// TIA Portal V20 export
FUNCTION_BLOCK "CallInterfaceSignals"   // FB38, LAD
TITLE = CallInterfaceSignals
AUTHOR : SICAR
FAMILY : Diag
VERSION : 1.0
// The block serves as a calling interface of the block “InterfaceSignalsBool“. The block is designed as function block in order to implement the block calls as multi-instances.
// stored: IsIECCheckEnabled true, MemoryReserve 100, SetENOAutomatically true
   VAR
      statReadValueHmi : Bool;   // HMI: Read value signal
      statSelectSignalsHmi : USInt := 1;   // HMI: Selected interface signals (1..16)
      statSelectSignalsOld { ExternalAccessible := 'False'; ExternalVisible := 'False'; ExternalWritable := 'False'} : USInt;   // Old value: Selected interface signals
      statRisEdgeReadName { ExternalAccessible := 'False'; ExternalVisible := 'False'; ExternalWritable := 'False'} : Bool;   // Rising edge
      statPosPulseReadName : Bool;   // Positive pulse
      statInterfaceSignalsHmi : Array[0..100] of "typeInterfaceSignalsHmi";   // HMI: Description, value and symbolic name
      instSignals1Left { ExternalAccessible := 'False'; ExternalVisible := 'False'; ExternalWritable := 'False'} : "LAF_InterfaceSignalsBool";   // interface signals screen 1 left
      instSignals1Right { ExternalAccessible := 'False'; ExternalVisible := 'False'; ExternalWritable := 'False'} : "LAF_InterfaceSignalsBool";   // interface signals screen 1 right
      instSignals2Left { ExternalAccessible := 'False'; ExternalVisible := 'False'; ExternalWritable := 'False'} : "LAF_InterfaceSignalsBool";   // interface signals screen 2 left
      instSignals2Right { ExternalAccessible := 'False'; ExternalVisible := 'False'; ExternalWritable := 'False'} : "LAF_InterfaceSignalsBool";   // interface signals screen 2 right
      instSignals3Left { ExternalAccessible := 'False'; ExternalVisible := 'False'; ExternalWritable := 'False'} : "LAF_InterfaceSignalsBool";   // interface signals screen 3 left
      instSignals3Right { ExternalAccessible := 'False'; ExternalVisible := 'False'; ExternalWritable := 'False'} : "LAF_InterfaceSignalsBool";   // interface signals screen 3 right
      instSignals4Left { ExternalAccessible := 'False'; ExternalVisible := 'False'; ExternalWritable := 'False'} : "LAF_InterfaceSignalsBool";   // interface signals screen 4 left
      instSignals4Right { ExternalAccessible := 'False'; ExternalVisible := 'False'; ExternalWritable := 'False'} : "LAF_InterfaceSignalsBool";   // interface signals screen 4 right
      instSignals5Left { ExternalAccessible := 'False'; ExternalVisible := 'False'; ExternalWritable := 'False'} : "LAF_InterfaceSignalsBool";   // interface signals screen 5 left
      instSignals5Right { ExternalAccessible := 'False'; ExternalVisible := 'False'; ExternalWritable := 'False'} : "LAF_InterfaceSignalsBool";   // interface signals screen 5 right
      instSignals6Left { S7_SetPoint := 'True'} : "LAF_InterfaceSignalsBool";   // interface signals screen 6 left
      instSignals6Right { S7_SetPoint := 'True'} : "LAF_InterfaceSignalsBool";   // interface signals screen 6 right
      instSignals7Left { S7_SetPoint := 'True'} : "LAF_InterfaceSignalsBool";   // interface signals screen 7 left
      instSignals7Right { S7_SetPoint := 'True'} : "LAF_InterfaceSignalsBool";   // interface signals screen 7 right
      instSignals8Left { S7_SetPoint := 'True'} : "LAF_InterfaceSignalsBool";   // interface signals screen 8 left
      instSignals8Right { S7_SetPoint := 'True'} : "LAF_InterfaceSignalsBool";   // interface signals screen 8 right
      instSignals9Left { S7_SetPoint := 'True'} : "LAF_InterfaceSignalsBool";   // interface signals screen 9 left
      instSignals9Right { S7_SetPoint := 'True'} : "LAF_InterfaceSignalsBool";   // interface signals screen 9 right
      instSignals10Left_ { S7_SetPoint := 'True'} : "LAF_InterfaceSignalsBool";   // interface signals screen 10 left
      instSignals10Right { S7_SetPoint := 'True'} : "LAF_InterfaceSignalsBool";   // interface signals screen 10 right
      instSignals11Left { S7_SetPoint := 'True'} : "LAF_InterfaceSignalsBool";   // interface signals screen 11 left
      instSignals11Right { S7_SetPoint := 'True'} : "LAF_InterfaceSignalsBool";   // interface signals screen 11 right
      instSignals12Left { S7_SetPoint := 'True'} : "LAF_InterfaceSignalsBool";   // interface signals screen 12 left
      instSignals12Right { S7_SetPoint := 'True'} : "LAF_InterfaceSignalsBool";   // interface signals screen 12 right
      instSignals13Left { S7_SetPoint := 'True'} : "LAF_InterfaceSignalsBool";   // interface signals screen 13 left
      instSignals13Right { S7_SetPoint := 'True'} : "LAF_InterfaceSignalsBool";   // interface signals screen 13 right
      instSignals14Left { S7_SetPoint := 'True'} : "LAF_InterfaceSignalsBool";   // interface signals screen 14 left
      instSignals14Right { S7_SetPoint := 'True'} : "LAF_InterfaceSignalsBool";   // interface signals screen 14 right
      instSignals15Left { S7_SetPoint := 'True'} : "LAF_InterfaceSignalsBool";   // interface signals screen 15 left
      instSignals15Right { S7_SetPoint := 'True'} : "LAF_InterfaceSignalsBool";   // interface signals screen 15 right
      instSignals16Left { S7_SetPoint := 'True'} : "LAF_InterfaceSignalsBool";   // interface signals screen 16 left
      instSignals16Right { S7_SetPoint := 'True'} : "LAF_InterfaceSignalsBool";   // interface signals screen 16 right
      instSignals17Left { S7_SetPoint := 'True'} : "LAF_InterfaceSignalsBool";   // interface signals screen 17 left
      instSignals17Right { S7_SetPoint := 'True'} : "LAF_InterfaceSignalsBool";   // interface signals screen 17 right
      instSignals18Left { S7_SetPoint := 'True'} : "LAF_InterfaceSignalsBool";   // interface signals screen 18 left
      instSignals18Right { S7_SetPoint := 'True'} : "LAF_InterfaceSignalsBool";   // interface signals screen 18 right
      instSignals19Left { S7_SetPoint := 'True'} : "LAF_InterfaceSignalsBool";   // interface signals screen 19 left
      instSignals19Right { S7_SetPoint := 'True'} : "LAF_InterfaceSignalsBool";   // interface signals screen 19 right
      instSignals20Left { S7_SetPoint := 'True'} : "LAF_InterfaceSignalsBool";   // interface signals screen 20 left
      instSignals20Right { S7_SetPoint := 'True'} : "LAF_InterfaceSignalsBool";   // interface signals screen 20 right
      instSignals21Left { S7_SetPoint := 'True'} : "LAF_InterfaceSignalsBool";   // interface signals screen 21 left
      instSignals21Right { S7_SetPoint := 'True'} : "LAF_InterfaceSignalsBool";   // interface signals screen 21 right
      instSignals22Left { S7_SetPoint := 'True'} : "LAF_InterfaceSignalsBool";   // interface signals screen 22 left
      instSignals22Right { S7_SetPoint := 'True'} : "LAF_InterfaceSignalsBool";   // interface signals screen 22 right
      instSignals23Left { S7_SetPoint := 'True'} : "LAF_InterfaceSignalsBool";   // interface signals screen 23 left
      instSignals23Right { S7_SetPoint := 'True'} : "LAF_InterfaceSignalsBool";   // interface signals screen 23 right
      instSignals24Left { S7_SetPoint := 'True'} : "LAF_InterfaceSignalsBool";   // interface signals screen 24 left
      instSignals24Right { S7_SetPoint := 'True'} : "LAF_InterfaceSignalsBool";   // interface signals screen 24 right
      instSignals25Left { S7_SetPoint := 'True'} : "LAF_InterfaceSignalsBool";   // interface signals screen 25 left
      instSignals25Right { S7_SetPoint := 'True'} : "LAF_InterfaceSignalsBool";   // interface signals screen 25 right
      instSignals26Left { S7_SetPoint := 'True'} : "LAF_InterfaceSignalsBool";   // interface signals screen 26 left
      instSignals26Right { S7_SetPoint := 'True'} : "LAF_InterfaceSignalsBool";   // interface signals screen 26 right
      instSignals27Left { S7_SetPoint := 'True'} : "LAF_InterfaceSignalsBool";   // interface signals screen 27 left
      instSignals27Right { S7_SetPoint := 'True'} : "LAF_InterfaceSignalsBool";   // interface signals screen 27 right
      instSignals28Left { S7_SetPoint := 'True'} : "LAF_InterfaceSignalsBool";   // interface signals screen 28 left
      instSignals28Right { S7_SetPoint := 'True'} : "LAF_InterfaceSignalsBool";   // interface signals screen 28 right
      instSignals29Left { S7_SetPoint := 'True'} : "LAF_InterfaceSignalsBool";   // interface signals screen 29 left
      instSignals29Right { S7_SetPoint := 'True'} : "LAF_InterfaceSignalsBool";   // interface signals screen 29 right
      instSignals30Left { S7_SetPoint := 'True'} : "LAF_InterfaceSignalsBool";   // interface signals screen 30 left
      instSignals30Right { S7_SetPoint := 'True'} : "LAF_InterfaceSignalsBool";   // interface signals screen 30 right
      instSignals31Left { S7_SetPoint := 'True'} : "LAF_InterfaceSignalsBool";   // interface signals screen 31 left
      instSignals31Right { S7_SetPoint := 'True'} : "LAF_InterfaceSignalsBool";   // interface signals screen 31 right
      instSignals32Left { S7_SetPoint := 'True'} : "LAF_InterfaceSignalsBool";   // interface signals screen 32 left
      instSignals32Right { S7_SetPoint := 'True'} : "LAF_InterfaceSignalsBool";   // interface signals screen 32 right
      instSignals33Left { S7_SetPoint := 'True'} : "LAF_InterfaceSignalsBool";   // interface signals screen 33 left
      instSignals33Right { S7_SetPoint := 'True'} : "LAF_InterfaceSignalsBool";   // interface signals screen 33 right
      instSignals34Left { S7_SetPoint := 'True'} : "LAF_InterfaceSignalsBool";   // interface signals screen 34 left
      instSignals34Right { S7_SetPoint := 'True'} : "LAF_InterfaceSignalsBool";   // interface signals screen 34 right
      instSignals35Left { S7_SetPoint := 'True'} : "LAF_InterfaceSignalsBool";   // interface signals screen 35 left
      instSignals35Right { S7_SetPoint := 'True'} : "LAF_InterfaceSignalsBool";   // interface signals screen 35 right
      instSignals36Left { S7_SetPoint := 'True'} : "LAF_InterfaceSignalsBool";   // interface signals screen 36 left
      instSignals36Right { S7_SetPoint := 'True'} : "LAF_InterfaceSignalsBool";   // interface signals screen 36 right
      instSignals37Left { S7_SetPoint := 'True'} : "LAF_InterfaceSignalsBool";   // interface signals screen 37 left
      instSignals37Right { S7_SetPoint := 'True'} : "LAF_InterfaceSignalsBool";   // interface signals screen 37 right
      instSignals38Left { S7_SetPoint := 'True'} : "LAF_InterfaceSignalsBool";   // interface signals screen 38 left
      instSignals38Right { S7_SetPoint := 'True'} : "LAF_InterfaceSignalsBool";   // interface signals screen 38 right
      instSignals39Left { S7_SetPoint := 'True'} : "LAF_InterfaceSignalsBool";   // interface signals screen 39 left
      instSignals39Right { S7_SetPoint := 'True'} : "LAF_InterfaceSignalsBool";   // interface signals screen 39 right
      instSignals40Left { S7_SetPoint := 'True'} : "LAF_InterfaceSignalsBool";   // interface signals screen 40 left
      instSignals40Right { S7_SetPoint := 'True'} : "LAF_InterfaceSignalsBool";   // interface signals screen 40 right
      instSignals41Left { S7_SetPoint := 'True'} : "LAF_InterfaceSignalsBool";   // interface signals screen 41 left
      instSignals41Right { S7_SetPoint := 'True'} : "LAF_InterfaceSignalsBool";   // interface signals screen 41 right
      instSignals42Left { S7_SetPoint := 'True'} : "LAF_InterfaceSignalsBool";   // interface signals screen 42 left
      instSignals42Right { S7_SetPoint := 'True'} : "LAF_InterfaceSignalsBool";   // interface signals screen 42 right
      instSignals43Left { S7_SetPoint := 'True'} : "LAF_InterfaceSignalsBool";   // interface signals screen 43 left
      instSignals43Right { S7_SetPoint := 'True'} : "LAF_InterfaceSignalsBool";   // interface signals screen 43 right
      instSignals44Left { S7_SetPoint := 'True'} : "LAF_InterfaceSignalsBool";   // interface signals screen 44 left
      instSignals44Right { S7_SetPoint := 'True'} : "LAF_InterfaceSignalsBool";   // interface signals screen 44 right
      instSignals45Left { S7_SetPoint := 'True'} : "LAF_InterfaceSignalsBool";   // interface signals screen 45 left
      instSignals45Right { S7_SetPoint := 'True'} : "LAF_InterfaceSignalsBool";   // interface signals screen 45 right
      instSignals46Left { S7_SetPoint := 'True'} : "LAF_InterfaceSignalsBool";   // interface signals screen 46 left
      instSignals46Right { S7_SetPoint := 'True'} : "LAF_InterfaceSignalsBool";   // interface signals screen 46 right
      instSignals47Left { S7_SetPoint := 'True'} : "LAF_InterfaceSignalsBool";   // interface signals screen 47 left
      instSignals47Right { S7_SetPoint := 'True'} : "LAF_InterfaceSignalsBool";   // interface signals screen 47 right
      instSignals48Left { S7_SetPoint := 'True'} : "LAF_InterfaceSignalsBool";   // interface signals screen 48 left
      instSignals48Right { S7_SetPoint := 'True'} : "LAF_InterfaceSignalsBool";   // interface signals screen 48 right
      instSignals49Left { S7_SetPoint := 'True'} : "LAF_InterfaceSignalsBool";   // interface signals screen 49 left
      instSignals49Right { S7_SetPoint := 'True'} : "LAF_InterfaceSignalsBool";   // interface signals screen 49 right
      instSignals50Left { S7_SetPoint := 'True'} : "LAF_InterfaceSignalsBool";   // interface signals screen 50 left
      instSignals50Right { S7_SetPoint := 'True'} : "LAF_InterfaceSignalsBool";   // interface signals screen 50 right
      instSignals51Left { S7_SetPoint := 'True'} : "LAF_InterfaceSignalsBool";   // interface signals screen 51 left
      instSignals51Right { S7_SetPoint := 'True'} : "LAF_InterfaceSignalsBool";   // interface signals screen 51 right
      instSignals52Left { S7_SetPoint := 'True'} : "LAF_InterfaceSignalsBool";   // interface signals screen 52 left
      instSignals52Right { S7_SetPoint := 'True'} : "LAF_InterfaceSignalsBool";   // interface signals screen 52 right
      instSignals53Left { S7_SetPoint := 'True'} : "LAF_InterfaceSignalsBool";   // interface signals screen 53 left
      instSignals53Right { S7_SetPoint := 'True'} : "LAF_InterfaceSignalsBool";   // interface signals screen 53 right
      instSignals54Left { S7_SetPoint := 'True'} : "LAF_InterfaceSignalsBool";   // interface signals screen 54 left
      instSignals54Right { S7_SetPoint := 'True'} : "LAF_InterfaceSignalsBool";   // interface signals screen 54 right
      instSignals55Left { S7_SetPoint := 'True'} : "LAF_InterfaceSignalsBool";   // interface signals screen 55 left
      instSignals55Right { S7_SetPoint := 'True'} : "LAF_InterfaceSignalsBool";   // interface signals screen 55 right
      instSignals56Left { S7_SetPoint := 'True'} : "LAF_InterfaceSignalsBool";   // interface signals screen 56 left
      instSignals56Right { S7_SetPoint := 'True'} : "LAF_InterfaceSignalsBool";   // interface signals screen 56 right
      instSignals57Left { S7_SetPoint := 'True'} : "LAF_InterfaceSignalsBool";   // interface signals screen 57 left
      instSignals57Right { S7_SetPoint := 'True'} : "LAF_InterfaceSignalsBool";   // interface signals screen 57 right
      instSignals58Left { S7_SetPoint := 'True'} : "LAF_InterfaceSignalsBool";   // interface signals screen 58 left
      instSignals58Right { S7_SetPoint := 'True'} : "LAF_InterfaceSignalsBool";   // interface signals screen 58 right
      instSignals59Left { S7_SetPoint := 'True'} : "LAF_InterfaceSignalsBool";   // interface signals screen 59 left
      instSignals59Right { S7_SetPoint := 'True'} : "LAF_InterfaceSignalsBool";   // interface signals screen 59 right
      instSignals60Left { S7_SetPoint := 'True'} : "LAF_InterfaceSignalsBool";   // interface signals screen 60 left
      instSignals60Right { S7_SetPoint := 'True'} : "LAF_InterfaceSignalsBool";   // interface signals screen 60 right
      instSignals61Left { S7_SetPoint := 'True'} : "LAF_InterfaceSignalsBool";   // interface signals screen 61 left
      instSignals61Right { S7_SetPoint := 'True'} : "LAF_InterfaceSignalsBool";   // interface signals screen 61 right
      instSignals62Left { S7_SetPoint := 'True'} : "LAF_InterfaceSignalsBool";   // interface signals screen 62 left
      instSignals62Right { S7_SetPoint := 'True'} : "LAF_InterfaceSignalsBool";   // interface signals screen 62 right
      instSignals63Left { S7_SetPoint := 'True'} : "LAF_InterfaceSignalsBool";   // interface signals screen 63 left
      instSignals63Right { S7_SetPoint := 'True'} : "LAF_InterfaceSignalsBool";   // interface signals screen 63 right
      instSignals64Left { S7_SetPoint := 'True'} : "LAF_InterfaceSignalsBool";   // interface signals screen 64 left
      instSignals64Right { S7_SetPoint := 'True'} : "LAF_InterfaceSignalsBool";   // interface signals screen 64 right
      instSignals65Left { S7_SetPoint := 'True'} : "LAF_InterfaceSignalsBool";   // interface signals screen 65 left
      instSignals65Right { S7_SetPoint := 'True'} : "LAF_InterfaceSignalsBool";   // interface signals screen 65 right
      instSignals66Left { S7_SetPoint := 'True'} : "LAF_InterfaceSignalsBool";   // interface signals screen 66 left
      instSignals66Right { S7_SetPoint := 'True'} : "LAF_InterfaceSignalsBool";   // interface signals screen 66 right
      instSignals67Left { S7_SetPoint := 'True'} : "LAF_InterfaceSignalsBool";   // interface signals screen 67 left
      instSignals67Right { S7_SetPoint := 'True'} : "LAF_InterfaceSignalsBool";   // interface signals screen 67 right
      instSignals68Left { S7_SetPoint := 'True'} : "LAF_InterfaceSignalsBool";   // interface signals screen 68 left
      instSignals68Right { S7_SetPoint := 'True'} : "LAF_InterfaceSignalsBool";   // interface signals screen 68 right
      instSignals69Left { S7_SetPoint := 'True'} : "LAF_InterfaceSignalsBool";   // interface signals screen 69 left
      instSignals69Right { S7_SetPoint := 'True'} : "LAF_InterfaceSignalsBool";   // interface signals screen 69 right
      instSignals70Left { S7_SetPoint := 'True'} : "LAF_InterfaceSignalsBool";   // interface signals screen 70 left
      instSignals70Right { S7_SetPoint := 'True'} : "LAF_InterfaceSignalsBool";   // interface signals screen 70 right
      instSignals71Left { S7_SetPoint := 'True'} : "LAF_InterfaceSignalsBool";   // interface signals screen 71 left
      instSignals71Right { S7_SetPoint := 'True'} : "LAF_InterfaceSignalsBool";   // interface signals screen 71 right
      instSignals72Left { S7_SetPoint := 'True'} : "LAF_InterfaceSignalsBool";   // interface signals screen 72 left
      instSignals72Right { S7_SetPoint := 'True'} : "LAF_InterfaceSignalsBool";   // interface signals screen 72 right
      instSignals73Left { S7_SetPoint := 'True'} : "LAF_InterfaceSignalsBool";   // interface signals screen 73 left
      instSignals73Right { S7_SetPoint := 'True'} : "LAF_InterfaceSignalsBool";   // interface signals screen 73 right
      instSignals74Left { S7_SetPoint := 'True'} : "LAF_InterfaceSignalsBool";   // interface signals screen 74 left
      instSignals74Right { S7_SetPoint := 'True'} : "LAF_InterfaceSignalsBool";   // interface signals screen 74 right
      instSignals75Left { S7_SetPoint := 'True'} : "LAF_InterfaceSignalsBool";   // interface signals screen 75 left
      instSignals75Right { S7_SetPoint := 'True'} : "LAF_InterfaceSignalsBool";   // interface signals screen 75 right
      instSignals76Left { S7_SetPoint := 'True'} : "LAF_InterfaceSignalsBool";   // interface signals screen 76 left
      instSignals76Right { S7_SetPoint := 'True'} : "LAF_InterfaceSignalsBool";   // interface signals screen 76 right
   END_VAR
   VAR_TEMP
      tempLoopCounter : DInt;   // temp. Loop Counter
   END_VAR
   VAR_TEMP   // added for the SCL form of the ladder/FBD networks
      _w1 : Bool;
   END_VAR
BEGIN

REGION Network 1: BLOCK INFO HEADER
   // SIEMENS AG / (c)Copyright 2023
   // ------------------------------------------------------------------------------
   // Title:            CallInterfaceSignals (FB38)
   // Comment/Function: The block serves as a calling interface of the block “InterfaceSignalsBool“. The block is designed as function block in order to implement the block calls as multi-instances. 
   // Library/Family:   Diag
   // Author:           SICAR
   // Tested with:      ---
   // Engineering:      TIA Portal V19
   // Restrictions:     -
   // Requirements:     ---
   // ------------------------------------------------------------------------------
   // Change log table:
   // Version  | Date       | Expert in charge       | Changes applied
   // ---------|------------|------------------------|------------------------------
   // 01.00.00 | 11.12.2023 | SICAR
   //                         First released version
END_REGION

REGION Network 2: DESCRIPTION
   // Function block and corresponding WinCC screen are prepared for 16 data sets (“InterfaceSignals01“ through .”InterfaceSignals16“) with 32 Boolean signals each.  
   // 
   // **PLC-Data types**   
   // 
   // * LSicar_typeInterfaceSignalsBool 
   // * LSicar _typeInterfaceSignals 
   // * typeInterfaceSignalsHmi 
   // 
   // **WinCC-Faceplate**  
   // 
   // <None> 
   // 
   // **WinCC Diagnostic screen**   
   // 
   // See: ..\Library Types\LSicar_InterfaceSignalsBool.pdf  
   // 
   // **Block call example** 
   // 
   // View in ladder-logic (LAD), without parameter settings.  
   // An executable program call is available in the “SICAR-Startup” project.  
   // 
   // **Calling interface**  
   // 
   // The block is be called once in the cyclic program.  
   // 
   // **Internally used „Extended instructions / blocks“**  
   // 
   // See: ..\Library Types\LSicar_InterfaceSignalsBool.pdf
END_REGION

REGION Network 3: Initialization Loop_1
   // Preset the loop index
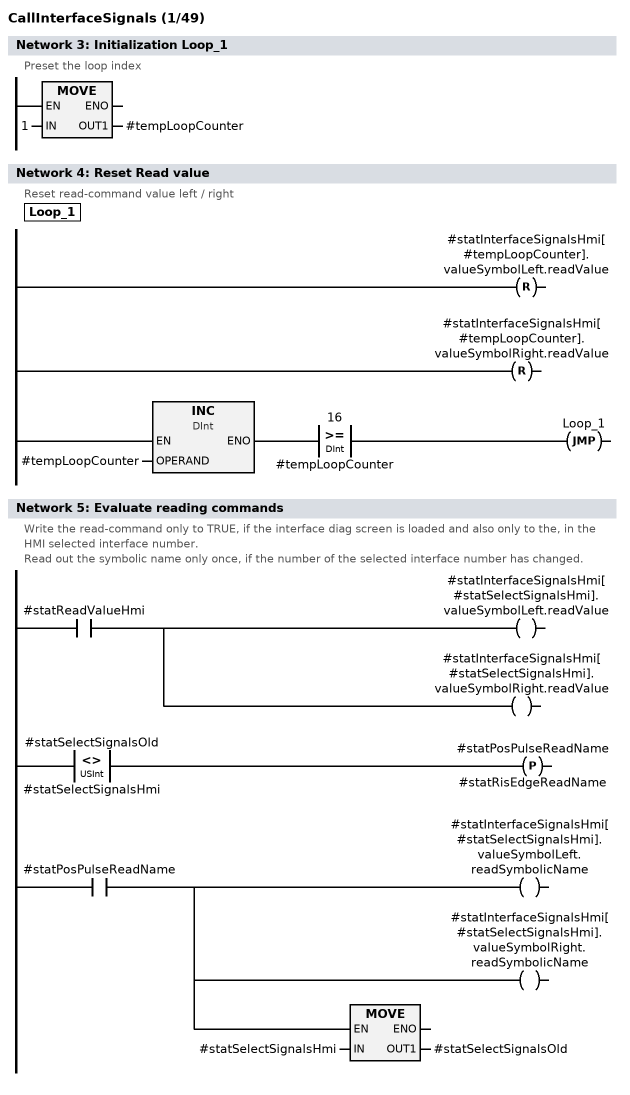
   RUNG wire#powerrail
      Move(in := 1, out1 => #tempLoopCounter)
   END_RUNG
   // the same network as SCL:
   #tempLoopCounter := 1;
END_REGION

REGION Network 4: Reset Read value
   // Reset read-command value left / right
   Label( Loop_1 )
   RUNG wire#powerrail
      R_Coil( #statInterfaceSignalsHmi[#tempLoopCounter].valueSymbolLeft.readValue )
   END_RUNG
   RUNG wire#powerrail
      R_Coil( #statInterfaceSignalsHmi[#tempLoopCounter].valueSymbolRight.readValue )
   END_RUNG
   RUNG wire#powerrail
      { S7_Templates := "DestType := DInt" } Inc( #tempLoopCounter )
      { S7_Templates := "SrcType := DInt" } GE_Contact(in1 := 16, in2 := #tempLoopCounter)
      JumpCoil( Loop_1 )
   END_RUNG
   // the same network as SCL:
   Loop_1:
   #statInterfaceSignalsHmi[#tempLoopCounter].valueSymbolLeft.readValue := FALSE;
   #statInterfaceSignalsHmi[#tempLoopCounter].valueSymbolRight.readValue := FALSE;
   #tempLoopCounter := #tempLoopCounter + 1;
   IF 16 >= #tempLoopCounter THEN GOTO Loop_1; END_IF;
END_REGION

REGION Network 5: Evaluate reading commands
   // Write the read-command only to TRUE, if the interface diag screen is loaded and also only to the, in the HMI selected interface number.
   // Read out the symbolic name only once, if the number of the selected interface number has changed.
   #statInterfaceSignalsHmi[#statSelectSignalsHmi].valueSymbolLeft.readValue := #statReadValueHmi;
   #statInterfaceSignalsHmi[#statSelectSignalsHmi].valueSymbolRight.readValue := #statReadValueHmi;
   #_w1 := #statSelectSignalsOld <> #statSelectSignalsHmi;
   #statPosPulseReadName := #_w1 AND NOT #statRisEdgeReadName;   // rising edge
   #statRisEdgeReadName := #_w1;
   #statInterfaceSignalsHmi[#statSelectSignalsHmi].valueSymbolLeft.readSymbolicName := #statPosPulseReadName;
   #statInterfaceSignalsHmi[#statSelectSignalsHmi].valueSymbolRight.readSymbolicName := #statPosPulseReadName;
   IF #statPosPulseReadName THEN #statSelectSignalsOld := #statSelectSignalsHmi; END_IF;
END_REGION

REGION Network 6: Interface Signals 01 BA030
   // Call the interface signals bool blocks of system tags
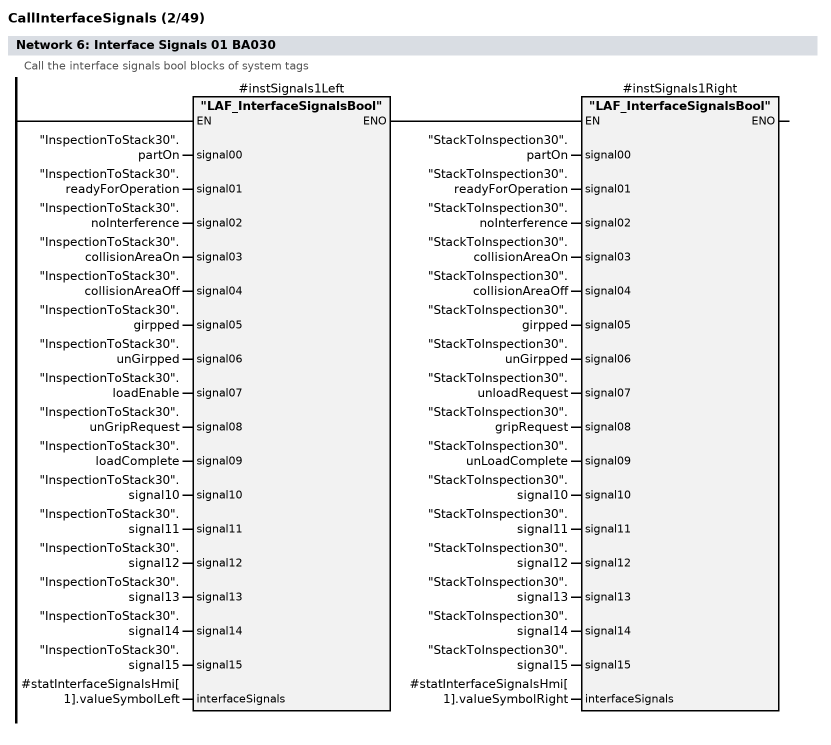
   RUNG wire#powerrail
      #instSignals1Left(signal00 := "InspectionToStack30".partOn, signal01 := "InspectionToStack30".readyForOperation, signal02 := "InspectionToStack30".noInterference, signal03 := "InspectionToStack30".collisionAreaOn, signal04 := "InspectionToStack30".collisionAreaOff, signal05 := "InspectionToStack30".girpped, signal06 := "InspectionToStack30".unGirpped, signal07 := "InspectionToStack30".loadEnable, signal08 := "InspectionToStack30".unGripRequest, signal09 := "InspectionToStack30".loadComplete, signal10 := "InspectionToStack30".signal10, signal11 := "InspectionToStack30".signal11, signal12 := "InspectionToStack30".signal12, signal13 := "InspectionToStack30".signal13, signal14 := "InspectionToStack30".signal14, signal15 := "InspectionToStack30".signal15, interfaceSignals := #statInterfaceSignalsHmi[1].valueSymbolLeft)
      #instSignals1Right(signal00 := "StackToInspection30".partOn, signal01 := "StackToInspection30".readyForOperation, signal02 := "StackToInspection30".noInterference, signal03 := "StackToInspection30".collisionAreaOn, signal04 := "StackToInspection30".collisionAreaOff, signal05 := "StackToInspection30".girpped, signal06 := "StackToInspection30".unGirpped, signal07 := "StackToInspection30".unloadRequest, signal08 := "StackToInspection30".gripRequest, signal09 := "StackToInspection30".unLoadComplete, signal10 := "StackToInspection30".signal10, signal11 := "StackToInspection30".signal11, signal12 := "StackToInspection30".signal12, signal13 := "StackToInspection30".signal13, signal14 := "StackToInspection30".signal14, signal15 := "StackToInspection30".signal15, interfaceSignals := #statInterfaceSignalsHmi[1].valueSymbolRight)
   END_RUNG
   // the same network as SCL:
   #instSignals1Left(signal00 := "InspectionToStack30".partOn,   // "LAF_InterfaceSignalsBool"
                     signal01 := "InspectionToStack30".readyForOperation,
                     signal02 := "InspectionToStack30".noInterference,
                     signal03 := "InspectionToStack30".collisionAreaOn,
                     signal04 := "InspectionToStack30".collisionAreaOff,
                     signal05 := "InspectionToStack30".girpped,
                     signal06 := "InspectionToStack30".unGirpped,
                     signal07 := "InspectionToStack30".loadEnable,
                     signal08 := "InspectionToStack30".unGripRequest,
                     signal09 := "InspectionToStack30".loadComplete,
                     signal10 := "InspectionToStack30".signal10,
                     signal11 := "InspectionToStack30".signal11,
                     signal12 := "InspectionToStack30".signal12,
                     signal13 := "InspectionToStack30".signal13,
                     signal14 := "InspectionToStack30".signal14,
                     signal15 := "InspectionToStack30".signal15,
                     interfaceSignals := #statInterfaceSignalsHmi[1].valueSymbolLeft,
                     ENO => #_w1);
   IF #_w1 THEN
       #instSignals1Right(signal00 := "StackToInspection30".partOn,   // "LAF_InterfaceSignalsBool"
                          signal01 := "StackToInspection30".readyForOperation,
                          signal02 := "StackToInspection30".noInterference,
                          signal03 := "StackToInspection30".collisionAreaOn,
                          signal04 := "StackToInspection30".collisionAreaOff,
                          signal05 := "StackToInspection30".girpped,
                          signal06 := "StackToInspection30".unGirpped,
                          signal07 := "StackToInspection30".unloadRequest,
                          signal08 := "StackToInspection30".gripRequest,
                          signal09 := "StackToInspection30".unLoadComplete,
                          signal10 := "StackToInspection30".signal10,
                          signal11 := "StackToInspection30".signal11,
                          signal12 := "StackToInspection30".signal12,
                          signal13 := "StackToInspection30".signal13,
                          signal14 := "StackToInspection30".signal14,
                          signal15 := "StackToInspection30".signal15,
                          interfaceSignals := #statInterfaceSignalsHmi[1].valueSymbolRight);
   END_IF;
END_REGION

REGION Network 7: Interface Signals 02 BA040
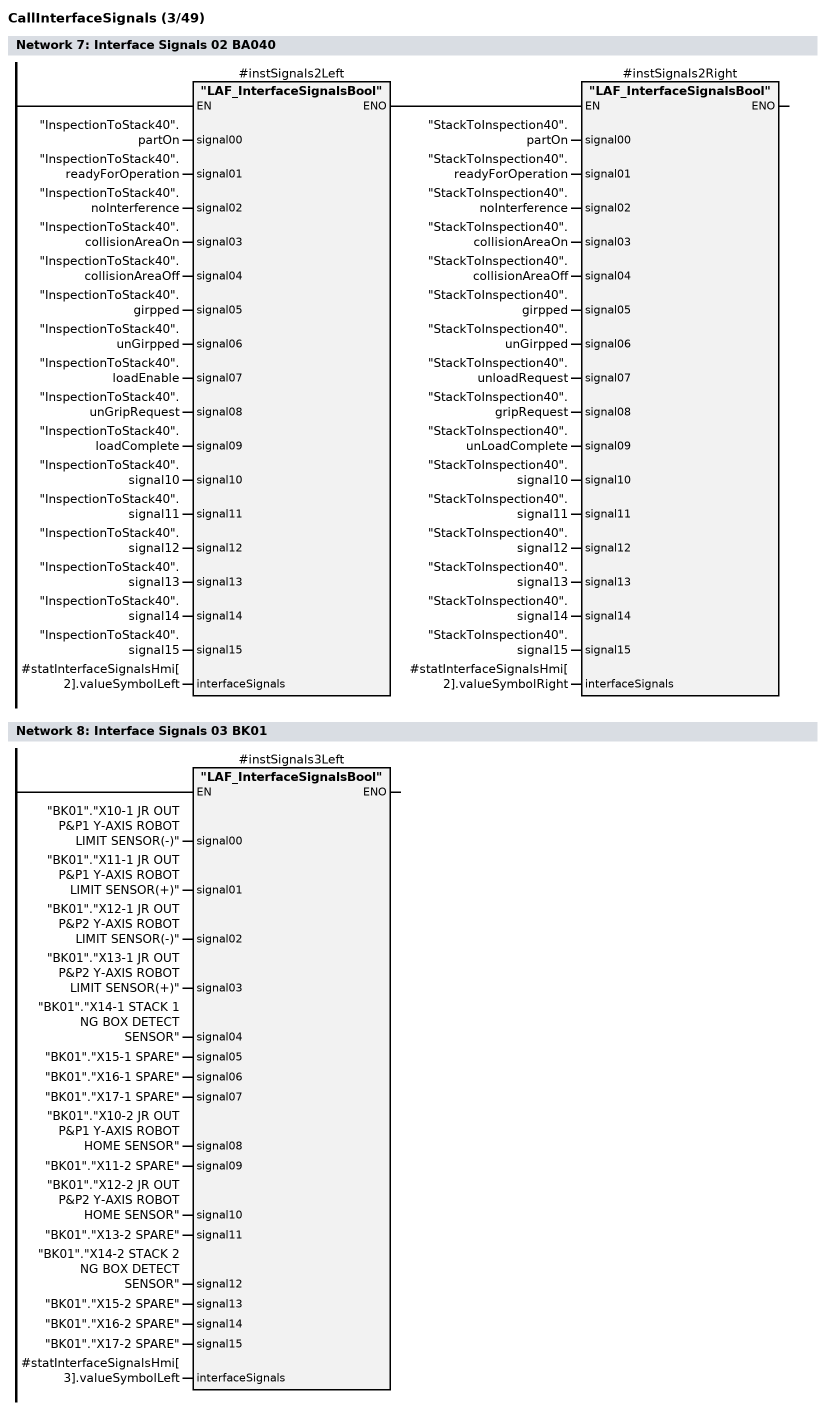
   RUNG wire#powerrail
      #instSignals2Left(signal00 := "InspectionToStack40".partOn, signal01 := "InspectionToStack40".readyForOperation, signal02 := "InspectionToStack40".noInterference, signal03 := "InspectionToStack40".collisionAreaOn, signal04 := "InspectionToStack40".collisionAreaOff, signal05 := "InspectionToStack40".girpped, signal06 := "InspectionToStack40".unGirpped, signal07 := "InspectionToStack40".loadEnable, signal08 := "InspectionToStack40".unGripRequest, signal09 := "InspectionToStack40".loadComplete, signal10 := "InspectionToStack40".signal10, signal11 := "InspectionToStack40".signal11, signal12 := "InspectionToStack40".signal12, signal13 := "InspectionToStack40".signal13, signal14 := "InspectionToStack40".signal14, signal15 := "InspectionToStack40".signal15, interfaceSignals := #statInterfaceSignalsHmi[2].valueSymbolLeft)
      #instSignals2Right(signal00 := "StackToInspection40".partOn, signal01 := "StackToInspection40".readyForOperation, signal02 := "StackToInspection40".noInterference, signal03 := "StackToInspection40".collisionAreaOn, signal04 := "StackToInspection40".collisionAreaOff, signal05 := "StackToInspection40".girpped, signal06 := "StackToInspection40".unGirpped, signal07 := "StackToInspection40".unloadRequest, signal08 := "StackToInspection40".gripRequest, signal09 := "StackToInspection40".unLoadComplete, signal10 := "StackToInspection40".signal10, signal11 := "StackToInspection40".signal11, signal12 := "StackToInspection40".signal12, signal13 := "StackToInspection40".signal13, signal14 := "StackToInspection40".signal14, signal15 := "StackToInspection40".signal15, interfaceSignals := #statInterfaceSignalsHmi[2].valueSymbolRight)
   END_RUNG
   // the same network as SCL:
   #instSignals2Left(signal00 := "InspectionToStack40".partOn,   // "LAF_InterfaceSignalsBool"
                     signal01 := "InspectionToStack40".readyForOperation,
                     signal02 := "InspectionToStack40".noInterference,
                     signal03 := "InspectionToStack40".collisionAreaOn,
                     signal04 := "InspectionToStack40".collisionAreaOff,
                     signal05 := "InspectionToStack40".girpped,
                     signal06 := "InspectionToStack40".unGirpped,
                     signal07 := "InspectionToStack40".loadEnable,
                     signal08 := "InspectionToStack40".unGripRequest,
                     signal09 := "InspectionToStack40".loadComplete,
                     signal10 := "InspectionToStack40".signal10,
                     signal11 := "InspectionToStack40".signal11,
                     signal12 := "InspectionToStack40".signal12,
                     signal13 := "InspectionToStack40".signal13,
                     signal14 := "InspectionToStack40".signal14,
                     signal15 := "InspectionToStack40".signal15,
                     interfaceSignals := #statInterfaceSignalsHmi[2].valueSymbolLeft,
                     ENO => #_w1);
   IF #_w1 THEN
       #instSignals2Right(signal00 := "StackToInspection40".partOn,   // "LAF_InterfaceSignalsBool"
                          signal01 := "StackToInspection40".readyForOperation,
                          signal02 := "StackToInspection40".noInterference,
                          signal03 := "StackToInspection40".collisionAreaOn,
                          signal04 := "StackToInspection40".collisionAreaOff,
                          signal05 := "StackToInspection40".girpped,
                          signal06 := "StackToInspection40".unGirpped,
                          signal07 := "StackToInspection40".unloadRequest,
                          signal08 := "StackToInspection40".gripRequest,
                          signal09 := "StackToInspection40".unLoadComplete,
                          signal10 := "StackToInspection40".signal10,
                          signal11 := "StackToInspection40".signal11,
                          signal12 := "StackToInspection40".signal12,
                          signal13 := "StackToInspection40".signal13,
                          signal14 := "StackToInspection40".signal14,
                          signal15 := "StackToInspection40".signal15,
                          interfaceSignals := #statInterfaceSignalsHmi[2].valueSymbolRight);
   END_IF;
END_REGION

REGION Network 8: Interface Signals 03 BK01
   RUNG wire#powerrail
      #instSignals3Left(signal00 := "BK01"."X10-1 JR OUT P&P1 Y-AXIS ROBOT LIMIT SENSOR(-)", signal01 := "BK01"."X11-1 JR OUT P&P1 Y-AXIS ROBOT LIMIT SENSOR(+)", signal02 := "BK01"."X12-1 JR OUT P&P2 Y-AXIS ROBOT LIMIT SENSOR(-)", signal03 := "BK01"."X13-1 JR OUT P&P2 Y-AXIS ROBOT LIMIT SENSOR(+)", signal04 := "BK01"."X14-1 STACK 1 NG BOX DETECT SENSOR", signal05 := "BK01"."X15-1 SPARE", signal06 := "BK01"."X16-1 SPARE", signal07 := "BK01"."X17-1 SPARE", signal08 := "BK01"."X10-2 JR OUT P&P1 Y-AXIS ROBOT HOME SENSOR", signal09 := "BK01"."X11-2 SPARE", signal10 := "BK01"."X12-2 JR OUT P&P2 Y-AXIS ROBOT HOME SENSOR", signal11 := "BK01"."X13-2 SPARE", signal12 := "BK01"."X14-2 STACK 2 NG BOX DETECT SENSOR", signal13 := "BK01"."X15-2 SPARE", signal14 := "BK01"."X16-2 SPARE", signal15 := "BK01"."X17-2 SPARE", interfaceSignals := #statInterfaceSignalsHmi[3].valueSymbolLeft)
   END_RUNG
   // the same network as SCL:
   #instSignals3Left(signal00 := "BK01"."X10-1 JR OUT P&P1 Y-AXIS ROBOT LIMIT SENSOR(-)",   // "LAF_InterfaceSignalsBool"
                     signal01 := "BK01"."X11-1 JR OUT P&P1 Y-AXIS ROBOT LIMIT SENSOR(+)",
                     signal02 := "BK01"."X12-1 JR OUT P&P2 Y-AXIS ROBOT LIMIT SENSOR(-)",
                     signal03 := "BK01"."X13-1 JR OUT P&P2 Y-AXIS ROBOT LIMIT SENSOR(+)",
                     signal04 := "BK01"."X14-1 STACK 1 NG BOX DETECT SENSOR",
                     signal05 := "BK01"."X15-1 SPARE",
                     signal06 := "BK01"."X16-1 SPARE",
                     signal07 := "BK01"."X17-1 SPARE",
                     signal08 := "BK01"."X10-2 JR OUT P&P1 Y-AXIS ROBOT HOME SENSOR",
                     signal09 := "BK01"."X11-2 SPARE",
                     signal10 := "BK01"."X12-2 JR OUT P&P2 Y-AXIS ROBOT HOME SENSOR",
                     signal11 := "BK01"."X13-2 SPARE",
                     signal12 := "BK01"."X14-2 STACK 2 NG BOX DETECT SENSOR",
                     signal13 := "BK01"."X15-2 SPARE",
                     signal14 := "BK01"."X16-2 SPARE",
                     signal15 := "BK01"."X17-2 SPARE",
                     interfaceSignals := #statInterfaceSignalsHmi[3].valueSymbolLeft);
END_REGION

REGION Network 9: Interface Signals 04 BK02
   // Call the interface signals bool blocks of opmode 4
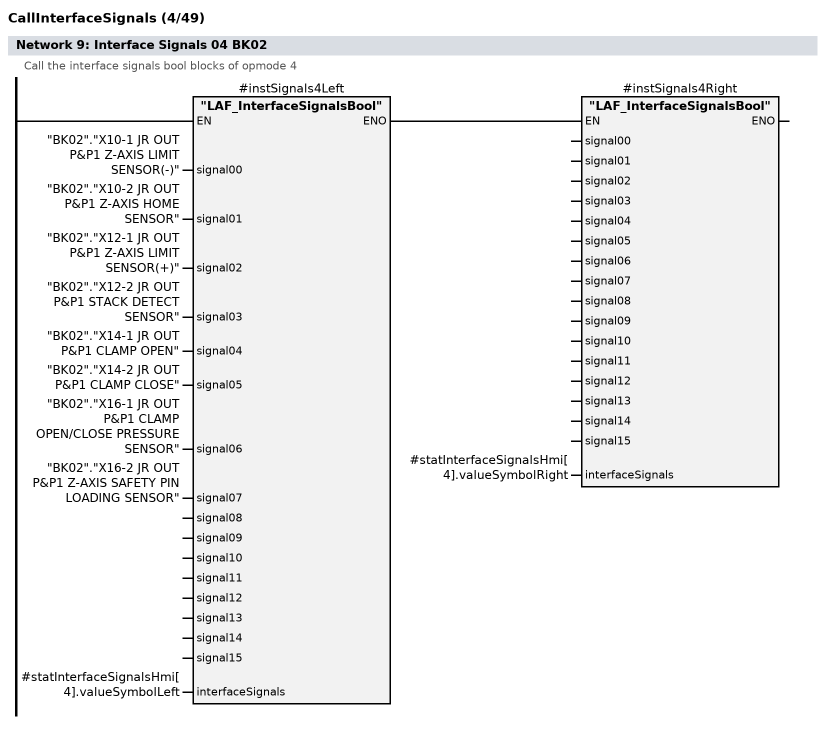
   RUNG wire#powerrail
      #instSignals4Left(signal00 := "BK02"."X10-1 JR OUT P&P1 Z-AXIS LIMIT SENSOR(-)", signal01 := "BK02"."X10-2 JR OUT P&P1 Z-AXIS HOME SENSOR", signal02 := "BK02"."X12-1 JR OUT P&P1 Z-AXIS LIMIT SENSOR(+)", signal03 := "BK02"."X12-2 JR OUT P&P1 STACK DETECT SENSOR", signal04 := "BK02"."X14-1 JR OUT P&P1 CLAMP OPEN", signal05 := "BK02"."X14-2 JR OUT P&P1 CLAMP CLOSE", signal06 := "BK02"."X16-1 JR OUT P&P1 CLAMP OPEN/CLOSE PRESSURE SENSOR", signal07 := "BK02"."X16-2 JR OUT P&P1 Z-AXIS SAFETY PIN LOADING SENSOR", signal08 :=, signal09 :=, signal10 :=, signal11 :=, signal12 :=, signal13 :=, signal14 :=, signal15 :=, interfaceSignals := #statInterfaceSignalsHmi[4].valueSymbolLeft)
      #instSignals4Right(signal00 :=, signal01 :=, signal02 :=, signal03 :=, signal04 :=, signal05 :=, signal06 :=, signal07 :=, signal08 :=, signal09 :=, signal10 :=, signal11 :=, signal12 :=, signal13 :=, signal14 :=, signal15 :=, interfaceSignals := #statInterfaceSignalsHmi[4].valueSymbolRight)
   END_RUNG
   // the same network as SCL:
   #instSignals4Left(signal00 := "BK02"."X10-1 JR OUT P&P1 Z-AXIS LIMIT SENSOR(-)",   // "LAF_InterfaceSignalsBool"
                     signal01 := "BK02"."X10-2 JR OUT P&P1 Z-AXIS HOME SENSOR",
                     signal02 := "BK02"."X12-1 JR OUT P&P1 Z-AXIS LIMIT SENSOR(+)",
                     signal03 := "BK02"."X12-2 JR OUT P&P1 STACK DETECT SENSOR",
                     signal04 := "BK02"."X14-1 JR OUT P&P1 CLAMP OPEN",
                     signal05 := "BK02"."X14-2 JR OUT P&P1 CLAMP CLOSE",
                     signal06 := "BK02"."X16-1 JR OUT P&P1 CLAMP OPEN/CLOSE PRESSURE SENSOR",
                     signal07 := "BK02"."X16-2 JR OUT P&P1 Z-AXIS SAFETY PIN LOADING SENSOR",
                     interfaceSignals := #statInterfaceSignalsHmi[4].valueSymbolLeft,
                     ENO => #_w1);
   IF #_w1 THEN
       #instSignals4Right(interfaceSignals := #statInterfaceSignalsHmi[4].valueSymbolRight);   // "LAF_InterfaceSignalsBool"
   END_IF;
END_REGION

REGION Network 10: Interface Signals 05 BK03
   // Call the interface signals bool blocks of opmode 4
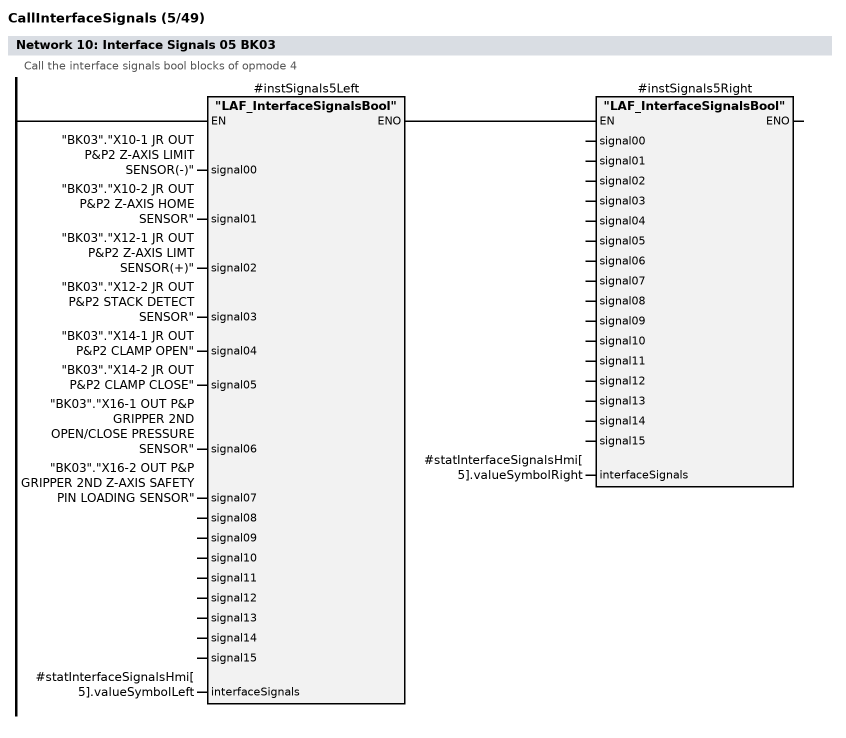
   RUNG wire#powerrail
      #instSignals5Left(signal00 := "BK03"."X10-1 JR OUT P&P2 Z-AXIS LIMIT SENSOR(-)", signal01 := "BK03"."X10-2 JR OUT P&P2 Z-AXIS HOME SENSOR", signal02 := "BK03"."X12-1 JR OUT P&P2 Z-AXIS LIMT SENSOR(+)", signal03 := "BK03"."X12-2 JR OUT P&P2 STACK DETECT SENSOR", signal04 := "BK03"."X14-1 JR OUT P&P2 CLAMP OPEN", signal05 := "BK03"."X14-2 JR OUT P&P2 CLAMP CLOSE", signal06 := "BK03"."X16-1 OUT P&P GRIPPER 2ND OPEN/CLOSE PRESSURE SENSOR", signal07 := "BK03"."X16-2 OUT P&P GRIPPER 2ND Z-AXIS SAFETY PIN LOADING SENSOR", signal08 :=, signal09 :=, signal10 :=, signal11 :=, signal12 :=, signal13 :=, signal14 :=, signal15 :=, interfaceSignals := #statInterfaceSignalsHmi[5].valueSymbolLeft)
      #instSignals5Right(signal00 :=, signal01 :=, signal02 :=, signal03 :=, signal04 :=, signal05 :=, signal06 :=, signal07 :=, signal08 :=, signal09 :=, signal10 :=, signal11 :=, signal12 :=, signal13 :=, signal14 :=, signal15 :=, interfaceSignals := #statInterfaceSignalsHmi[5].valueSymbolRight)
   END_RUNG
   // the same network as SCL:
   #instSignals5Left(signal00 := "BK03"."X10-1 JR OUT P&P2 Z-AXIS LIMIT SENSOR(-)",   // "LAF_InterfaceSignalsBool"
                     signal01 := "BK03"."X10-2 JR OUT P&P2 Z-AXIS HOME SENSOR",
                     signal02 := "BK03"."X12-1 JR OUT P&P2 Z-AXIS LIMT SENSOR(+)",
                     signal03 := "BK03"."X12-2 JR OUT P&P2 STACK DETECT SENSOR",
                     signal04 := "BK03"."X14-1 JR OUT P&P2 CLAMP OPEN",
                     signal05 := "BK03"."X14-2 JR OUT P&P2 CLAMP CLOSE",
                     signal06 := "BK03"."X16-1 OUT P&P GRIPPER 2ND OPEN/CLOSE PRESSURE SENSOR",
                     signal07 := "BK03"."X16-2 OUT P&P GRIPPER 2ND Z-AXIS SAFETY PIN LOADING SENSOR",
                     interfaceSignals := #statInterfaceSignalsHmi[5].valueSymbolLeft,
                     ENO => #_w1);
   IF #_w1 THEN
       #instSignals5Right(interfaceSignals := #statInterfaceSignalsHmi[5].valueSymbolRight);   // "LAF_InterfaceSignalsBool"
   END_IF;
END_REGION

REGION Network 11: Interface Signals 06 BK 04
   // Call the interface signals bool blocks
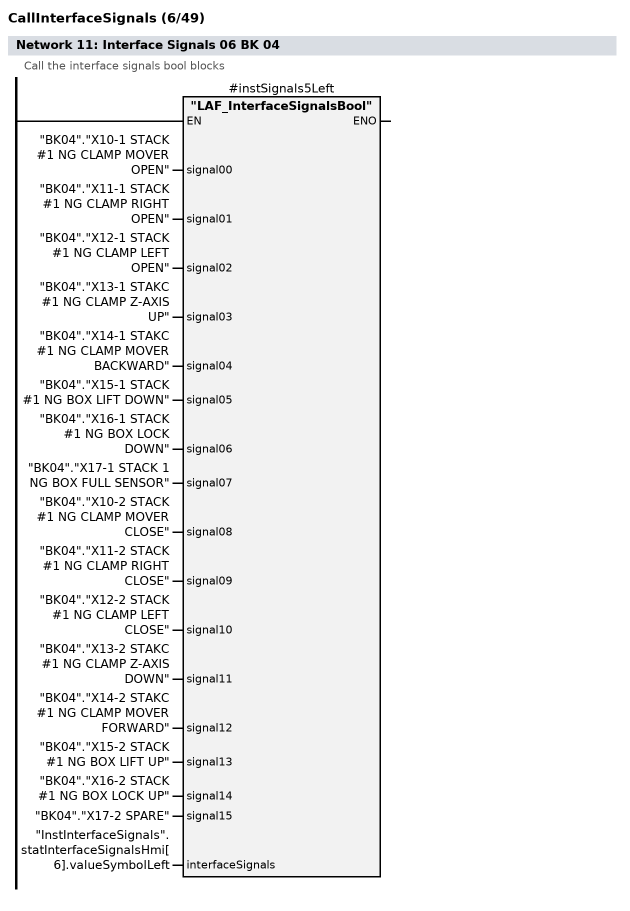
   RUNG wire#powerrail
      #instSignals5Left(signal00 := "BK04"."X10-1 STACK #1 NG CLAMP MOVER OPEN", signal01 := "BK04"."X11-1 STACK #1 NG CLAMP RIGHT OPEN", signal02 := "BK04"."X12-1 STACK #1 NG CLAMP LEFT OPEN", signal03 := "BK04"."X13-1 STAKC #1 NG CLAMP Z-AXIS UP", signal04 := "BK04"."X14-1 STAKC #1 NG CLAMP MOVER BACKWARD", signal05 := "BK04"."X15-1 STACK #1 NG BOX LIFT DOWN", signal06 := "BK04"."X16-1 STACK #1 NG BOX LOCK DOWN", signal07 := "BK04"."X17-1 STACK 1 NG BOX FULL SENSOR", signal08 := "BK04"."X10-2 STACK #1 NG CLAMP MOVER CLOSE", signal09 := "BK04"."X11-2 STACK #1 NG CLAMP RIGHT CLOSE", signal10 := "BK04"."X12-2 STACK #1 NG CLAMP LEFT CLOSE", signal11 := "BK04"."X13-2 STAKC #1 NG CLAMP Z-AXIS DOWN", signal12 := "BK04"."X14-2 STAKC #1 NG CLAMP MOVER FORWARD", signal13 := "BK04"."X15-2 STACK #1 NG BOX LIFT UP", signal14 := "BK04"."X16-2 STACK #1 NG BOX LOCK UP", signal15 := "BK04"."X17-2 SPARE", interfaceSignals := "InstInterfaceSignals".statInterfaceSignalsHmi[6].valueSymbolLeft)
   END_RUNG
   // the same network as SCL:
   #instSignals5Left(signal00 := "BK04"."X10-1 STACK #1 NG CLAMP MOVER OPEN",   // "LAF_InterfaceSignalsBool"
                     signal01 := "BK04"."X11-1 STACK #1 NG CLAMP RIGHT OPEN",
                     signal02 := "BK04"."X12-1 STACK #1 NG CLAMP LEFT OPEN",
                     signal03 := "BK04"."X13-1 STAKC #1 NG CLAMP Z-AXIS UP",
                     signal04 := "BK04"."X14-1 STAKC #1 NG CLAMP MOVER BACKWARD",
                     signal05 := "BK04"."X15-1 STACK #1 NG BOX LIFT DOWN",
                     signal06 := "BK04"."X16-1 STACK #1 NG BOX LOCK DOWN",
                     signal07 := "BK04"."X17-1 STACK 1 NG BOX FULL SENSOR",
                     signal08 := "BK04"."X10-2 STACK #1 NG CLAMP MOVER CLOSE",
                     signal09 := "BK04"."X11-2 STACK #1 NG CLAMP RIGHT CLOSE",
                     signal10 := "BK04"."X12-2 STACK #1 NG CLAMP LEFT CLOSE",
                     signal11 := "BK04"."X13-2 STAKC #1 NG CLAMP Z-AXIS DOWN",
                     signal12 := "BK04"."X14-2 STAKC #1 NG CLAMP MOVER FORWARD",
                     signal13 := "BK04"."X15-2 STACK #1 NG BOX LIFT UP",
                     signal14 := "BK04"."X16-2 STACK #1 NG BOX LOCK UP",
                     signal15 := "BK04"."X17-2 SPARE",
                     interfaceSignals := "InstInterfaceSignals".statInterfaceSignalsHmi[6].valueSymbolLeft);
END_REGION

REGION Network 12: Interface Signals 07 BK5
   // Call the interface signals bool blocks
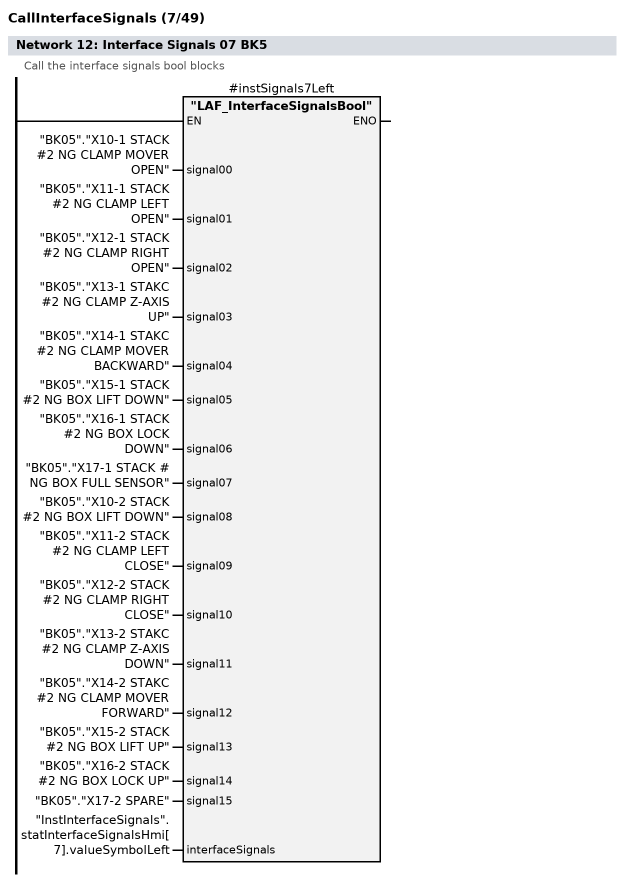
   RUNG wire#powerrail
      #instSignals7Left(signal00 := "BK05"."X10-1 STACK #2 NG CLAMP MOVER OPEN", signal01 := "BK05"."X11-1 STACK #2 NG CLAMP LEFT OPEN", signal02 := "BK05"."X12-1 STACK #2 NG CLAMP RIGHT OPEN", signal03 := "BK05"."X13-1 STAKC #2 NG CLAMP Z-AXIS UP", signal04 := "BK05"."X14-1 STAKC #2 NG CLAMP MOVER BACKWARD", signal05 := "BK05"."X15-1 STACK #2 NG BOX LIFT DOWN", signal06 := "BK05"."X16-1 STACK #2 NG BOX LOCK DOWN", signal07 := "BK05"."X17-1 STACK # NG BOX FULL SENSOR", signal08 := "BK05"."X10-2 STACK #2 NG BOX LIFT DOWN", signal09 := "BK05"."X11-2 STACK #2 NG CLAMP LEFT CLOSE", signal10 := "BK05"."X12-2 STACK #2 NG CLAMP RIGHT CLOSE", signal11 := "BK05"."X13-2 STAKC #2 NG CLAMP Z-AXIS DOWN", signal12 := "BK05"."X14-2 STAKC #2 NG CLAMP MOVER FORWARD", signal13 := "BK05"."X15-2 STACK #2 NG BOX LIFT UP", signal14 := "BK05"."X16-2 STACK #2 NG BOX LOCK UP", signal15 := "BK05"."X17-2 SPARE", interfaceSignals := "InstInterfaceSignals".statInterfaceSignalsHmi[7].valueSymbolLeft)
   END_RUNG
   // the same network as SCL:
   #instSignals7Left(signal00 := "BK05"."X10-1 STACK #2 NG CLAMP MOVER OPEN",   // "LAF_InterfaceSignalsBool"
                     signal01 := "BK05"."X11-1 STACK #2 NG CLAMP LEFT OPEN",
                     signal02 := "BK05"."X12-1 STACK #2 NG CLAMP RIGHT OPEN",
                     signal03 := "BK05"."X13-1 STAKC #2 NG CLAMP Z-AXIS UP",
                     signal04 := "BK05"."X14-1 STAKC #2 NG CLAMP MOVER BACKWARD",
                     signal05 := "BK05"."X15-1 STACK #2 NG BOX LIFT DOWN",
                     signal06 := "BK05"."X16-1 STACK #2 NG BOX LOCK DOWN",
                     signal07 := "BK05"."X17-1 STACK # NG BOX FULL SENSOR",
                     signal08 := "BK05"."X10-2 STACK #2 NG BOX LIFT DOWN",
                     signal09 := "BK05"."X11-2 STACK #2 NG CLAMP LEFT CLOSE",
                     signal10 := "BK05"."X12-2 STACK #2 NG CLAMP RIGHT CLOSE",
                     signal11 := "BK05"."X13-2 STAKC #2 NG CLAMP Z-AXIS DOWN",
                     signal12 := "BK05"."X14-2 STAKC #2 NG CLAMP MOVER FORWARD",
                     signal13 := "BK05"."X15-2 STACK #2 NG BOX LIFT UP",
                     signal14 := "BK05"."X16-2 STACK #2 NG BOX LOCK UP",
                     signal15 := "BK05"."X17-2 SPARE",
                     interfaceSignals := "InstInterfaceSignals".statInterfaceSignalsHmi[7].valueSymbolLeft);
END_REGION

REGION Network 13: Interface Signals 08 BK6
   // Call the interface signals bool blocks
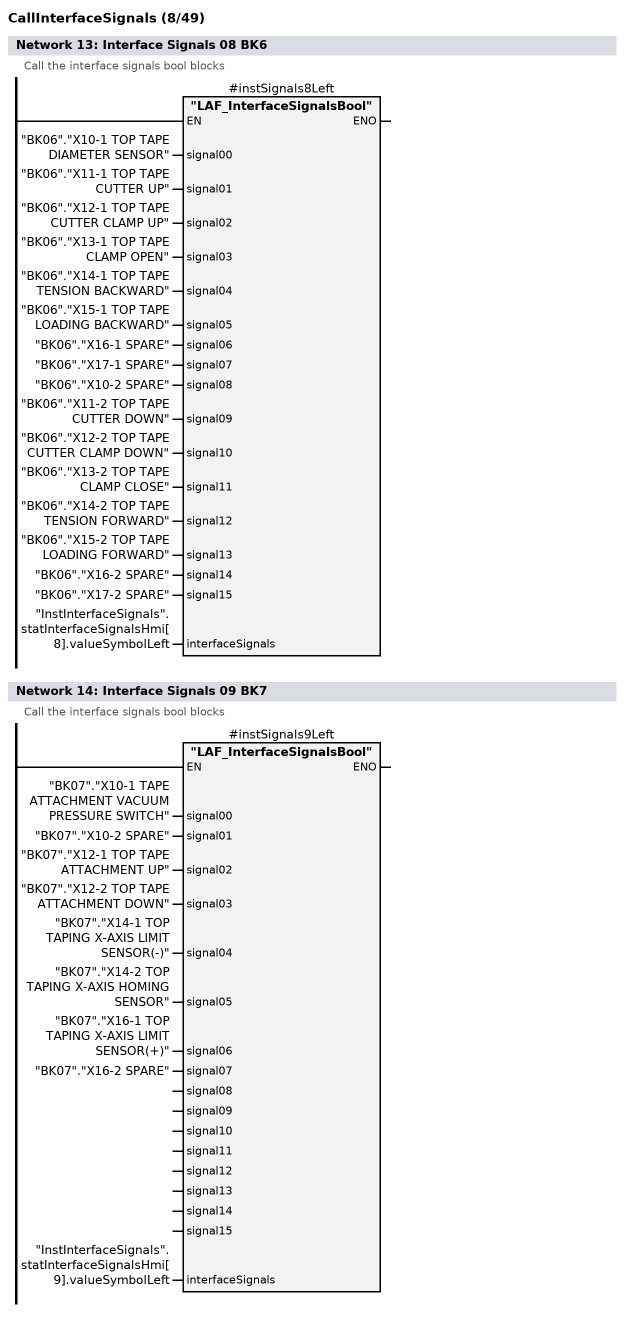
   RUNG wire#powerrail
      #instSignals8Left(signal00 := "BK06"."X10-1 TOP TAPE DIAMETER SENSOR", signal01 := "BK06"."X11-1 TOP TAPE CUTTER UP", signal02 := "BK06"."X12-1 TOP TAPE CUTTER CLAMP UP", signal03 := "BK06"."X13-1 TOP TAPE CLAMP OPEN", signal04 := "BK06"."X14-1 TOP TAPE TENSION BACKWARD", signal05 := "BK06"."X15-1 TOP TAPE LOADING BACKWARD", signal06 := "BK06"."X16-1 SPARE", signal07 := "BK06"."X17-1 SPARE", signal08 := "BK06"."X10-2 SPARE", signal09 := "BK06"."X11-2 TOP TAPE CUTTER DOWN", signal10 := "BK06"."X12-2 TOP TAPE CUTTER CLAMP DOWN", signal11 := "BK06"."X13-2 TOP TAPE CLAMP CLOSE", signal12 := "BK06"."X14-2 TOP TAPE TENSION FORWARD", signal13 := "BK06"."X15-2 TOP TAPE LOADING FORWARD", signal14 := "BK06"."X16-2 SPARE", signal15 := "BK06"."X17-2 SPARE", interfaceSignals := "InstInterfaceSignals".statInterfaceSignalsHmi[8].valueSymbolLeft)
   END_RUNG
   // the same network as SCL:
   #instSignals8Left(signal00 := "BK06"."X10-1 TOP TAPE DIAMETER SENSOR",   // "LAF_InterfaceSignalsBool"
                     signal01 := "BK06"."X11-1 TOP TAPE CUTTER UP",
                     signal02 := "BK06"."X12-1 TOP TAPE CUTTER CLAMP UP",
                     signal03 := "BK06"."X13-1 TOP TAPE CLAMP OPEN",
                     signal04 := "BK06"."X14-1 TOP TAPE TENSION BACKWARD",
                     signal05 := "BK06"."X15-1 TOP TAPE LOADING BACKWARD",
                     signal06 := "BK06"."X16-1 SPARE",
                     signal07 := "BK06"."X17-1 SPARE",
                     signal08 := "BK06"."X10-2 SPARE",
                     signal09 := "BK06"."X11-2 TOP TAPE CUTTER DOWN",
                     signal10 := "BK06"."X12-2 TOP TAPE CUTTER CLAMP DOWN",
                     signal11 := "BK06"."X13-2 TOP TAPE CLAMP CLOSE",
                     signal12 := "BK06"."X14-2 TOP TAPE TENSION FORWARD",
                     signal13 := "BK06"."X15-2 TOP TAPE LOADING FORWARD",
                     signal14 := "BK06"."X16-2 SPARE",
                     signal15 := "BK06"."X17-2 SPARE",
                     interfaceSignals := "InstInterfaceSignals".statInterfaceSignalsHmi[8].valueSymbolLeft);
END_REGION

REGION Network 14: Interface Signals 09 BK7
   // Call the interface signals bool blocks
   RUNG wire#powerrail
      #instSignals9Left(signal00 := "BK07"."X10-1 TAPE ATTACHMENT VACUUM PRESSURE SWITCH", signal01 := "BK07"."X10-2 SPARE", signal02 := "BK07"."X12-1 TOP TAPE ATTACHMENT UP", signal03 := "BK07"."X12-2 TOP TAPE ATTACHMENT DOWN", signal04 := "BK07"."X14-1 TOP TAPING X-AXIS LIMIT SENSOR(-)", signal05 := "BK07"."X14-2 TOP TAPING X-AXIS HOMING SENSOR", signal06 := "BK07"."X16-1 TOP TAPING X-AXIS LIMIT SENSOR(+)", signal07 := "BK07"."X16-2 SPARE", signal08 :=, signal09 :=, signal10 :=, signal11 :=, signal12 :=, signal13 :=, signal14 :=, signal15 :=, interfaceSignals := "InstInterfaceSignals".statInterfaceSignalsHmi[9].valueSymbolLeft)
   END_RUNG
   // the same network as SCL:
   #instSignals9Left(signal00 := "BK07"."X10-1 TAPE ATTACHMENT VACUUM PRESSURE SWITCH",   // "LAF_InterfaceSignalsBool"
                     signal01 := "BK07"."X10-2 SPARE",
                     signal02 := "BK07"."X12-1 TOP TAPE ATTACHMENT UP",
                     signal03 := "BK07"."X12-2 TOP TAPE ATTACHMENT DOWN",
                     signal04 := "BK07"."X14-1 TOP TAPING X-AXIS LIMIT SENSOR(-)",
                     signal05 := "BK07"."X14-2 TOP TAPING X-AXIS HOMING SENSOR",
                     signal06 := "BK07"."X16-1 TOP TAPING X-AXIS LIMIT SENSOR(+)",
                     signal07 := "BK07"."X16-2 SPARE",
                     interfaceSignals := "InstInterfaceSignals".statInterfaceSignalsHmi[9].valueSymbolLeft);
END_REGION

REGION Network 15: Interface Signals 10 BK8
   // Call the interface signals bool blocks
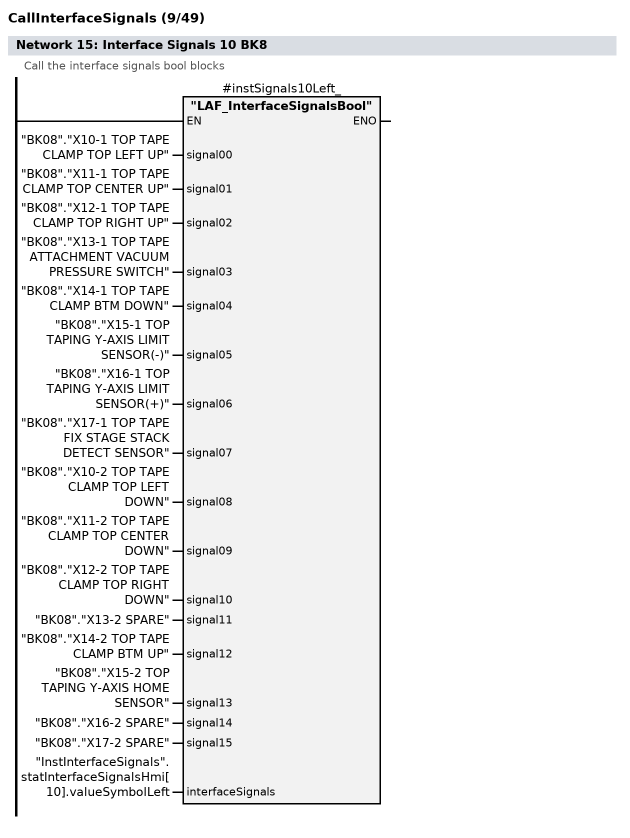
   RUNG wire#powerrail
      #instSignals10Left_(signal00 := "BK08"."X10-1 TOP TAPE CLAMP TOP LEFT UP", signal01 := "BK08"."X11-1 TOP TAPE CLAMP TOP CENTER UP", signal02 := "BK08"."X12-1 TOP TAPE CLAMP TOP RIGHT UP", signal03 := "BK08"."X13-1 TOP TAPE ATTACHMENT VACUUM PRESSURE SWITCH", signal04 := "BK08"."X14-1 TOP TAPE CLAMP BTM DOWN", signal05 := "BK08"."X15-1 TOP TAPING Y-AXIS LIMIT SENSOR(-)", signal06 := "BK08"."X16-1 TOP TAPING Y-AXIS LIMIT SENSOR(+)", signal07 := "BK08"."X17-1 TOP TAPE FIX STAGE STACK DETECT SENSOR", signal08 := "BK08"."X10-2 TOP TAPE CLAMP TOP LEFT DOWN", signal09 := "BK08"."X11-2 TOP TAPE CLAMP TOP CENTER DOWN", signal10 := "BK08"."X12-2 TOP TAPE CLAMP TOP RIGHT DOWN", signal11 := "BK08"."X13-2 SPARE", signal12 := "BK08"."X14-2 TOP TAPE CLAMP BTM UP", signal13 := "BK08"."X15-2 TOP TAPING Y-AXIS HOME SENSOR", signal14 := "BK08"."X16-2 SPARE", signal15 := "BK08"."X17-2 SPARE", interfaceSignals := "InstInterfaceSignals".statInterfaceSignalsHmi[10].valueSymbolLeft)
   END_RUNG
   // the same network as SCL:
   #instSignals10Left_(signal00 := "BK08"."X10-1 TOP TAPE CLAMP TOP LEFT UP",   // "LAF_InterfaceSignalsBool"
                       signal01 := "BK08"."X11-1 TOP TAPE CLAMP TOP CENTER UP",
                       signal02 := "BK08"."X12-1 TOP TAPE CLAMP TOP RIGHT UP",
                       signal03 := "BK08"."X13-1 TOP TAPE ATTACHMENT VACUUM PRESSURE SWITCH",
                       signal04 := "BK08"."X14-1 TOP TAPE CLAMP BTM DOWN",
                       signal05 := "BK08"."X15-1 TOP TAPING Y-AXIS LIMIT SENSOR(-)",
                       signal06 := "BK08"."X16-1 TOP TAPING Y-AXIS LIMIT SENSOR(+)",
                       signal07 := "BK08"."X17-1 TOP TAPE FIX STAGE STACK DETECT SENSOR",
                       signal08 := "BK08"."X10-2 TOP TAPE CLAMP TOP LEFT DOWN",
                       signal09 := "BK08"."X11-2 TOP TAPE CLAMP TOP CENTER DOWN",
                       signal10 := "BK08"."X12-2 TOP TAPE CLAMP TOP RIGHT DOWN",
                       signal11 := "BK08"."X13-2 SPARE",
                       signal12 := "BK08"."X14-2 TOP TAPE CLAMP BTM UP",
                       signal13 := "BK08"."X15-2 TOP TAPING Y-AXIS HOME SENSOR",
                       signal14 := "BK08"."X16-2 SPARE",
                       signal15 := "BK08"."X17-2 SPARE",
                       interfaceSignals := "InstInterfaceSignals".statInterfaceSignalsHmi[10].valueSymbolLeft);
END_REGION

REGION Network 16: Interface Signals 11 BK9
   // Call the interface signals bool blocks
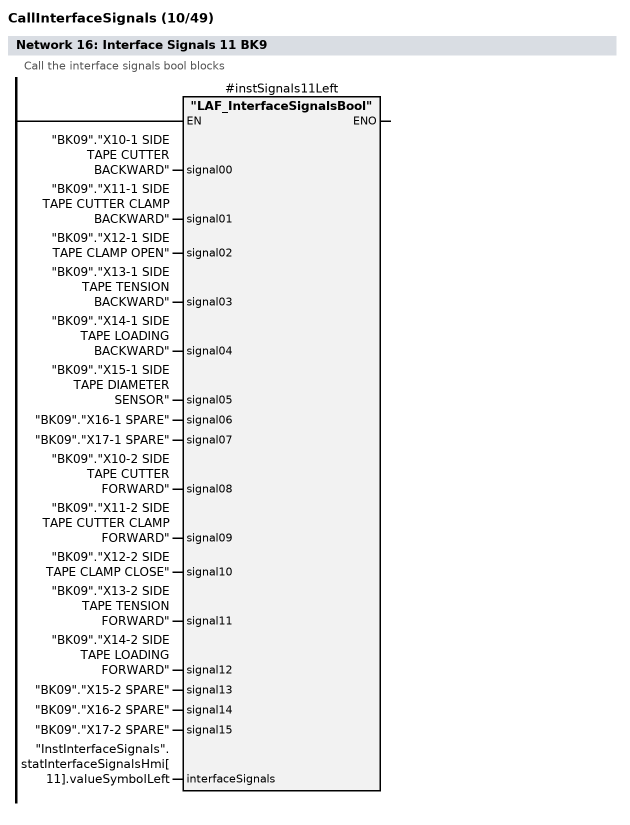
   RUNG wire#powerrail
      #instSignals11Left(signal00 := "BK09"."X10-1 SIDE TAPE CUTTER BACKWARD", signal01 := "BK09"."X11-1 SIDE TAPE CUTTER CLAMP BACKWARD", signal02 := "BK09"."X12-1 SIDE TAPE CLAMP OPEN", signal03 := "BK09"."X13-1 SIDE TAPE TENSION BACKWARD", signal04 := "BK09"."X14-1 SIDE TAPE LOADING BACKWARD", signal05 := "BK09"."X15-1 SIDE TAPE DIAMETER SENSOR", signal06 := "BK09"."X16-1 SPARE", signal07 := "BK09"."X17-1 SPARE", signal08 := "BK09"."X10-2 SIDE TAPE CUTTER FORWARD", signal09 := "BK09"."X11-2 SIDE TAPE CUTTER CLAMP FORWARD", signal10 := "BK09"."X12-2 SIDE TAPE CLAMP CLOSE", signal11 := "BK09"."X13-2 SIDE TAPE TENSION FORWARD", signal12 := "BK09"."X14-2 SIDE TAPE LOADING FORWARD", signal13 := "BK09"."X15-2 SPARE", signal14 := "BK09"."X16-2 SPARE", signal15 := "BK09"."X17-2 SPARE", interfaceSignals := "InstInterfaceSignals".statInterfaceSignalsHmi[11].valueSymbolLeft)
   END_RUNG
   // the same network as SCL:
   #instSignals11Left(signal00 := "BK09"."X10-1 SIDE TAPE CUTTER BACKWARD",   // "LAF_InterfaceSignalsBool"
                      signal01 := "BK09"."X11-1 SIDE TAPE CUTTER CLAMP BACKWARD",
                      signal02 := "BK09"."X12-1 SIDE TAPE CLAMP OPEN",
                      signal03 := "BK09"."X13-1 SIDE TAPE TENSION BACKWARD",
                      signal04 := "BK09"."X14-1 SIDE TAPE LOADING BACKWARD",
                      signal05 := "BK09"."X15-1 SIDE TAPE DIAMETER SENSOR",
                      signal06 := "BK09"."X16-1 SPARE",
                      signal07 := "BK09"."X17-1 SPARE",
                      signal08 := "BK09"."X10-2 SIDE TAPE CUTTER FORWARD",
                      signal09 := "BK09"."X11-2 SIDE TAPE CUTTER CLAMP FORWARD",
                      signal10 := "BK09"."X12-2 SIDE TAPE CLAMP CLOSE",
                      signal11 := "BK09"."X13-2 SIDE TAPE TENSION FORWARD",
                      signal12 := "BK09"."X14-2 SIDE TAPE LOADING FORWARD",
                      signal13 := "BK09"."X15-2 SPARE",
                      signal14 := "BK09"."X16-2 SPARE",
                      signal15 := "BK09"."X17-2 SPARE",
                      interfaceSignals := "InstInterfaceSignals".statInterfaceSignalsHmi[11].valueSymbolLeft);
END_REGION

REGION Network 17: Interface Signals 12 BK10
   // Call the interface signals bool blocks
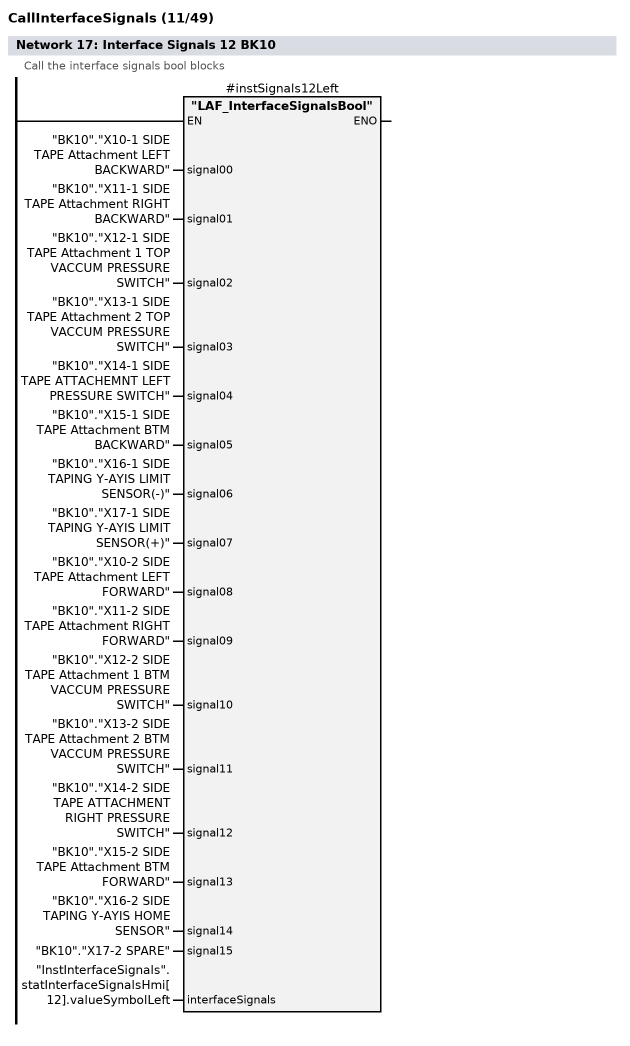
   RUNG wire#powerrail
      #instSignals12Left(signal00 := "BK10"."X10-1 SIDE TAPE Attachment LEFT BACKWARD", signal01 := "BK10"."X11-1 SIDE TAPE Attachment RIGHT BACKWARD", signal02 := "BK10"."X12-1 SIDE TAPE Attachment 1 TOP VACCUM PRESSURE SWITCH", signal03 := "BK10"."X13-1 SIDE TAPE Attachment 2 TOP VACCUM PRESSURE SWITCH", signal04 := "BK10"."X14-1 SIDE TAPE ATTACHEMNT LEFT PRESSURE SWITCH", signal05 := "BK10"."X15-1 SIDE TAPE Attachment BTM BACKWARD", signal06 := "BK10"."X16-1 SIDE TAPING Y-AYIS LIMIT SENSOR(-)", signal07 := "BK10"."X17-1 SIDE TAPING Y-AYIS LIMIT SENSOR(+)", signal08 := "BK10"."X10-2 SIDE TAPE Attachment LEFT FORWARD", signal09 := "BK10"."X11-2 SIDE TAPE Attachment RIGHT FORWARD", signal10 := "BK10"."X12-2 SIDE TAPE Attachment 1 BTM VACCUM PRESSURE SWITCH", signal11 := "BK10"."X13-2 SIDE TAPE Attachment 2 BTM VACCUM PRESSURE SWITCH", signal12 := "BK10"."X14-2 SIDE TAPE ATTACHMENT RIGHT PRESSURE SWITCH", signal13 := "BK10"."X15-2 SIDE TAPE Attachment BTM FORWARD", signal14 := "BK10"."X16-2 SIDE TAPING Y-AYIS HOME SENSOR", signal15 := "BK10"."X17-2 SPARE", interfaceSignals := "InstInterfaceSignals".statInterfaceSignalsHmi[12].valueSymbolLeft)
   END_RUNG
   // the same network as SCL:
   #instSignals12Left(signal00 := "BK10"."X10-1 SIDE TAPE Attachment LEFT BACKWARD",   // "LAF_InterfaceSignalsBool"
                      signal01 := "BK10"."X11-1 SIDE TAPE Attachment RIGHT BACKWARD",
                      signal02 := "BK10"."X12-1 SIDE TAPE Attachment 1 TOP VACCUM PRESSURE SWITCH",
                      signal03 := "BK10"."X13-1 SIDE TAPE Attachment 2 TOP VACCUM PRESSURE SWITCH",
                      signal04 := "BK10"."X14-1 SIDE TAPE ATTACHEMNT LEFT PRESSURE SWITCH",
                      signal05 := "BK10"."X15-1 SIDE TAPE Attachment BTM BACKWARD",
                      signal06 := "BK10"."X16-1 SIDE TAPING Y-AYIS LIMIT SENSOR(-)",
                      signal07 := "BK10"."X17-1 SIDE TAPING Y-AYIS LIMIT SENSOR(+)",
                      signal08 := "BK10"."X10-2 SIDE TAPE Attachment LEFT FORWARD",
                      signal09 := "BK10"."X11-2 SIDE TAPE Attachment RIGHT FORWARD",
                      signal10 := "BK10"."X12-2 SIDE TAPE Attachment 1 BTM VACCUM PRESSURE SWITCH",
                      signal11 := "BK10"."X13-2 SIDE TAPE Attachment 2 BTM VACCUM PRESSURE SWITCH",
                      signal12 := "BK10"."X14-2 SIDE TAPE ATTACHMENT RIGHT PRESSURE SWITCH",
                      signal13 := "BK10"."X15-2 SIDE TAPE Attachment BTM FORWARD",
                      signal14 := "BK10"."X16-2 SIDE TAPING Y-AYIS HOME SENSOR",
                      signal15 := "BK10"."X17-2 SPARE",
                      interfaceSignals := "InstInterfaceSignals".statInterfaceSignalsHmi[12].valueSymbolLeft);
END_REGION

REGION Network 18: Interface Signals 13 BK11
   // Call the interface signals bool blocks
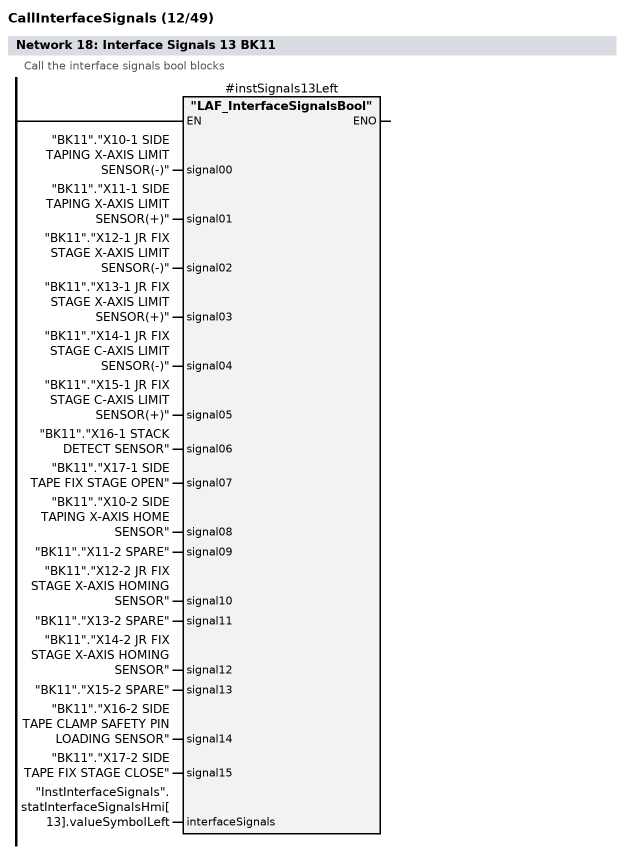
   RUNG wire#powerrail
      #instSignals13Left(signal00 := "BK11"."X10-1 SIDE TAPING X-AXIS LIMIT SENSOR(-)", signal01 := "BK11"."X11-1 SIDE TAPING X-AXIS LIMIT SENSOR(+)", signal02 := "BK11"."X12-1 JR FIX STAGE X-AXIS LIMIT SENSOR(-)", signal03 := "BK11"."X13-1 JR FIX STAGE X-AXIS LIMIT SENSOR(+)", signal04 := "BK11"."X14-1 JR FIX STAGE C-AXIS LIMIT SENSOR(-)", signal05 := "BK11"."X15-1 JR FIX STAGE C-AXIS LIMIT SENSOR(+)", signal06 := "BK11"."X16-1 STACK DETECT SENSOR", signal07 := "BK11"."X17-1 SIDE TAPE FIX STAGE OPEN", signal08 := "BK11"."X10-2 SIDE TAPING X-AXIS HOME SENSOR", signal09 := "BK11"."X11-2 SPARE", signal10 := "BK11"."X12-2 JR FIX STAGE X-AXIS HOMING SENSOR", signal11 := "BK11"."X13-2 SPARE", signal12 := "BK11"."X14-2 JR FIX STAGE X-AXIS HOMING SENSOR", signal13 := "BK11"."X15-2 SPARE", signal14 := "BK11"."X16-2 SIDE TAPE CLAMP SAFETY PIN LOADING SENSOR", signal15 := "BK11"."X17-2 SIDE TAPE FIX STAGE CLOSE", interfaceSignals := "InstInterfaceSignals".statInterfaceSignalsHmi[13].valueSymbolLeft)
   END_RUNG
   // the same network as SCL:
   #instSignals13Left(signal00 := "BK11"."X10-1 SIDE TAPING X-AXIS LIMIT SENSOR(-)",   // "LAF_InterfaceSignalsBool"
                      signal01 := "BK11"."X11-1 SIDE TAPING X-AXIS LIMIT SENSOR(+)",
                      signal02 := "BK11"."X12-1 JR FIX STAGE X-AXIS LIMIT SENSOR(-)",
                      signal03 := "BK11"."X13-1 JR FIX STAGE X-AXIS LIMIT SENSOR(+)",
                      signal04 := "BK11"."X14-1 JR FIX STAGE C-AXIS LIMIT SENSOR(-)",
                      signal05 := "BK11"."X15-1 JR FIX STAGE C-AXIS LIMIT SENSOR(+)",
                      signal06 := "BK11"."X16-1 STACK DETECT SENSOR",
                      signal07 := "BK11"."X17-1 SIDE TAPE FIX STAGE OPEN",
                      signal08 := "BK11"."X10-2 SIDE TAPING X-AXIS HOME SENSOR",
                      signal09 := "BK11"."X11-2 SPARE",
                      signal10 := "BK11"."X12-2 JR FIX STAGE X-AXIS HOMING SENSOR",
                      signal11 := "BK11"."X13-2 SPARE",
                      signal12 := "BK11"."X14-2 JR FIX STAGE X-AXIS HOMING SENSOR",
                      signal13 := "BK11"."X15-2 SPARE",
                      signal14 := "BK11"."X16-2 SIDE TAPE CLAMP SAFETY PIN LOADING SENSOR",
                      signal15 := "BK11"."X17-2 SIDE TAPE FIX STAGE CLOSE",
                      interfaceSignals := "InstInterfaceSignals".statInterfaceSignalsHmi[13].valueSymbolLeft);
END_REGION

REGION Network 19: Interface Signals 14 BK12
   // Call the interface signals bool blocks
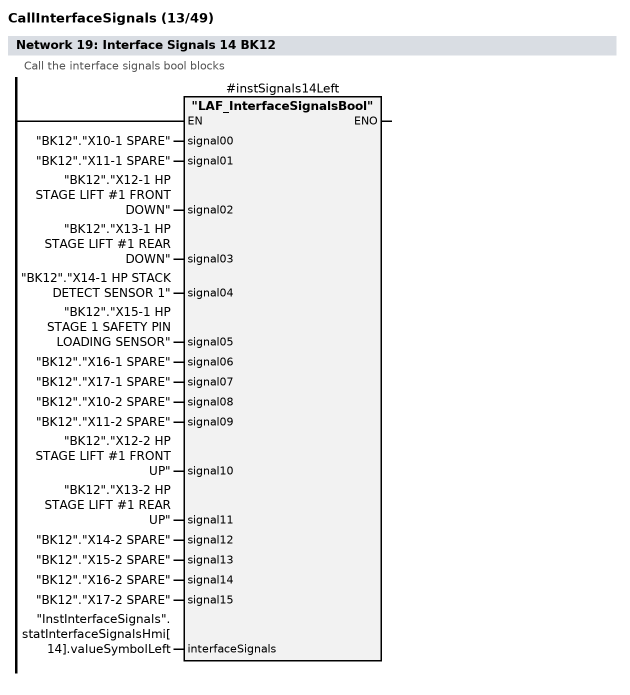
   RUNG wire#powerrail
      #instSignals14Left(signal00 := "BK12"."X10-1 SPARE", signal01 := "BK12"."X11-1 SPARE", signal02 := "BK12"."X12-1 HP STAGE LIFT #1 FRONT DOWN", signal03 := "BK12"."X13-1 HP STAGE LIFT #1 REAR DOWN", signal04 := "BK12"."X14-1 HP STACK DETECT SENSOR 1", signal05 := "BK12"."X15-1 HP STAGE 1 SAFETY PIN LOADING SENSOR", signal06 := "BK12"."X16-1 SPARE", signal07 := "BK12"."X17-1 SPARE", signal08 := "BK12"."X10-2 SPARE", signal09 := "BK12"."X11-2 SPARE", signal10 := "BK12"."X12-2 HP STAGE LIFT #1 FRONT UP", signal11 := "BK12"."X13-2 HP STAGE LIFT #1 REAR UP", signal12 := "BK12"."X14-2 SPARE", signal13 := "BK12"."X15-2 SPARE", signal14 := "BK12"."X16-2 SPARE", signal15 := "BK12"."X17-2 SPARE", interfaceSignals := "InstInterfaceSignals".statInterfaceSignalsHmi[14].valueSymbolLeft)
   END_RUNG
   // the same network as SCL:
   #instSignals14Left(signal00 := "BK12"."X10-1 SPARE",   // "LAF_InterfaceSignalsBool"
                      signal01 := "BK12"."X11-1 SPARE",
                      signal02 := "BK12"."X12-1 HP STAGE LIFT #1 FRONT DOWN",
                      signal03 := "BK12"."X13-1 HP STAGE LIFT #1 REAR DOWN",
                      signal04 := "BK12"."X14-1 HP STACK DETECT SENSOR 1",
                      signal05 := "BK12"."X15-1 HP STAGE 1 SAFETY PIN LOADING SENSOR",
                      signal06 := "BK12"."X16-1 SPARE",
                      signal07 := "BK12"."X17-1 SPARE",
                      signal08 := "BK12"."X10-2 SPARE",
                      signal09 := "BK12"."X11-2 SPARE",
                      signal10 := "BK12"."X12-2 HP STAGE LIFT #1 FRONT UP",
                      signal11 := "BK12"."X13-2 HP STAGE LIFT #1 REAR UP",
                      signal12 := "BK12"."X14-2 SPARE",
                      signal13 := "BK12"."X15-2 SPARE",
                      signal14 := "BK12"."X16-2 SPARE",
                      signal15 := "BK12"."X17-2 SPARE",
                      interfaceSignals := "InstInterfaceSignals".statInterfaceSignalsHmi[14].valueSymbolLeft);
END_REGION

REGION Network 20: Interface Signals 15 BK13
   // Call the interface signals bool blocks
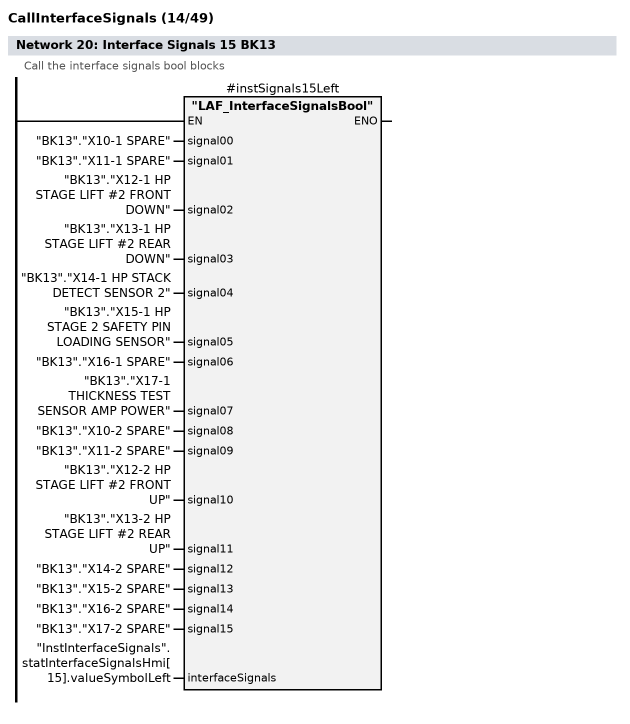
   RUNG wire#powerrail
      #instSignals15Left(signal00 := "BK13"."X10-1 SPARE", signal01 := "BK13"."X11-1 SPARE", signal02 := "BK13"."X12-1 HP STAGE LIFT #2 FRONT DOWN", signal03 := "BK13"."X13-1 HP STAGE LIFT #2 REAR DOWN", signal04 := "BK13"."X14-1 HP STACK DETECT SENSOR 2", signal05 := "BK13"."X15-1 HP STAGE 2 SAFETY PIN LOADING SENSOR", signal06 := "BK13"."X16-1 SPARE", signal07 := "BK13"."X17-1 THICKNESS TEST SENSOR AMP POWER", signal08 := "BK13"."X10-2 SPARE", signal09 := "BK13"."X11-2 SPARE", signal10 := "BK13"."X12-2 HP STAGE LIFT #2 FRONT UP", signal11 := "BK13"."X13-2 HP STAGE LIFT #2 REAR UP", signal12 := "BK13"."X14-2 SPARE", signal13 := "BK13"."X15-2 SPARE", signal14 := "BK13"."X16-2 SPARE", signal15 := "BK13"."X17-2 SPARE", interfaceSignals := "InstInterfaceSignals".statInterfaceSignalsHmi[15].valueSymbolLeft)
   END_RUNG
   // the same network as SCL:
   #instSignals15Left(signal00 := "BK13"."X10-1 SPARE",   // "LAF_InterfaceSignalsBool"
                      signal01 := "BK13"."X11-1 SPARE",
                      signal02 := "BK13"."X12-1 HP STAGE LIFT #2 FRONT DOWN",
                      signal03 := "BK13"."X13-1 HP STAGE LIFT #2 REAR DOWN",
                      signal04 := "BK13"."X14-1 HP STACK DETECT SENSOR 2",
                      signal05 := "BK13"."X15-1 HP STAGE 2 SAFETY PIN LOADING SENSOR",
                      signal06 := "BK13"."X16-1 SPARE",
                      signal07 := "BK13"."X17-1 THICKNESS TEST SENSOR AMP POWER",
                      signal08 := "BK13"."X10-2 SPARE",
                      signal09 := "BK13"."X11-2 SPARE",
                      signal10 := "BK13"."X12-2 HP STAGE LIFT #2 FRONT UP",
                      signal11 := "BK13"."X13-2 HP STAGE LIFT #2 REAR UP",
                      signal12 := "BK13"."X14-2 SPARE",
                      signal13 := "BK13"."X15-2 SPARE",
                      signal14 := "BK13"."X16-2 SPARE",
                      signal15 := "BK13"."X17-2 SPARE",
                      interfaceSignals := "InstInterfaceSignals".statInterfaceSignalsHmi[15].valueSymbolLeft);
END_REGION

REGION Network 21: Interface Signals 16 BK14
   // Call the interface signals bool blocks
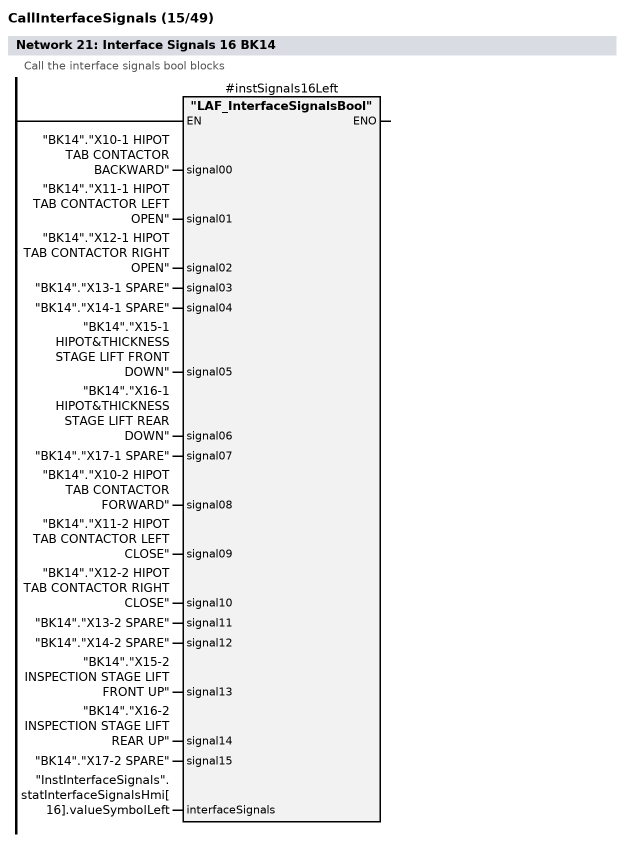
   RUNG wire#powerrail
      #instSignals16Left(signal00 := "BK14"."X10-1 HIPOT TAB CONTACTOR BACKWARD", signal01 := "BK14"."X11-1 HIPOT TAB CONTACTOR LEFT OPEN", signal02 := "BK14"."X12-1 HIPOT TAB CONTACTOR RIGHT OPEN", signal03 := "BK14"."X13-1 SPARE", signal04 := "BK14"."X14-1 SPARE", signal05 := "BK14"."X15-1 HIPOT&THICKNESS STAGE LIFT FRONT DOWN", signal06 := "BK14"."X16-1 HIPOT&THICKNESS STAGE LIFT REAR DOWN", signal07 := "BK14"."X17-1 SPARE", signal08 := "BK14"."X10-2 HIPOT TAB CONTACTOR FORWARD", signal09 := "BK14"."X11-2 HIPOT TAB CONTACTOR LEFT CLOSE", signal10 := "BK14"."X12-2 HIPOT TAB CONTACTOR RIGHT CLOSE", signal11 := "BK14"."X13-2 SPARE", signal12 := "BK14"."X14-2 SPARE", signal13 := "BK14"."X15-2 INSPECTION STAGE LIFT FRONT UP", signal14 := "BK14"."X16-2 INSPECTION STAGE LIFT REAR UP", signal15 := "BK14"."X17-2 SPARE", interfaceSignals := "InstInterfaceSignals".statInterfaceSignalsHmi[16].valueSymbolLeft)
   END_RUNG
   // the same network as SCL:
   #instSignals16Left(signal00 := "BK14"."X10-1 HIPOT TAB CONTACTOR BACKWARD",   // "LAF_InterfaceSignalsBool"
                      signal01 := "BK14"."X11-1 HIPOT TAB CONTACTOR LEFT OPEN",
                      signal02 := "BK14"."X12-1 HIPOT TAB CONTACTOR RIGHT OPEN",
                      signal03 := "BK14"."X13-1 SPARE",
                      signal04 := "BK14"."X14-1 SPARE",
                      signal05 := "BK14"."X15-1 HIPOT&THICKNESS STAGE LIFT FRONT DOWN",
                      signal06 := "BK14"."X16-1 HIPOT&THICKNESS STAGE LIFT REAR DOWN",
                      signal07 := "BK14"."X17-1 SPARE",
                      signal08 := "BK14"."X10-2 HIPOT TAB CONTACTOR FORWARD",
                      signal09 := "BK14"."X11-2 HIPOT TAB CONTACTOR LEFT CLOSE",
                      signal10 := "BK14"."X12-2 HIPOT TAB CONTACTOR RIGHT CLOSE",
                      signal11 := "BK14"."X13-2 SPARE",
                      signal12 := "BK14"."X14-2 SPARE",
                      signal13 := "BK14"."X15-2 INSPECTION STAGE LIFT FRONT UP",
                      signal14 := "BK14"."X16-2 INSPECTION STAGE LIFT REAR UP",
                      signal15 := "BK14"."X17-2 SPARE",
                      interfaceSignals := "InstInterfaceSignals".statInterfaceSignalsHmi[16].valueSymbolLeft);
END_REGION

REGION Network 22: Interface Signals 17 BK15
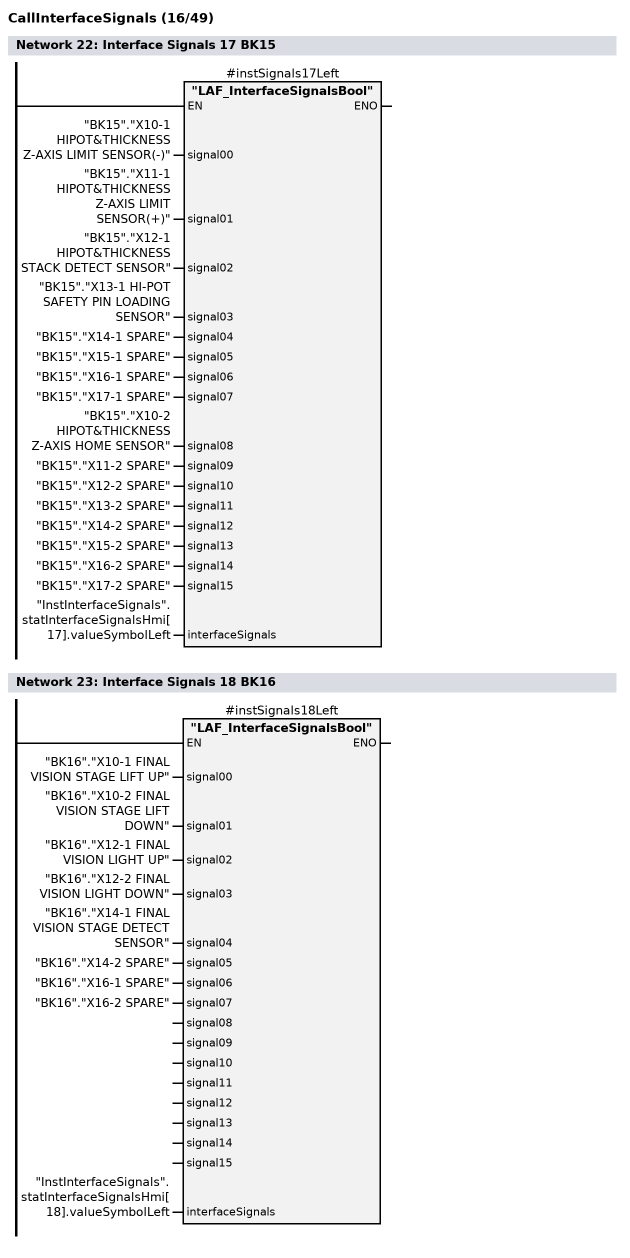
   RUNG wire#powerrail
      #instSignals17Left(signal00 := "BK15"."X10-1 HIPOT&THICKNESS Z-AXIS LIMIT SENSOR(-)", signal01 := "BK15"."X11-1 HIPOT&THICKNESS Z-AXIS LIMIT SENSOR(+)", signal02 := "BK15"."X12-1 HIPOT&THICKNESS STACK DETECT SENSOR", signal03 := "BK15"."X13-1 HI-POT SAFETY PIN LOADING SENSOR", signal04 := "BK15"."X14-1 SPARE", signal05 := "BK15"."X15-1 SPARE", signal06 := "BK15"."X16-1 SPARE", signal07 := "BK15"."X17-1 SPARE", signal08 := "BK15"."X10-2 HIPOT&THICKNESS Z-AXIS HOME SENSOR", signal09 := "BK15"."X11-2 SPARE", signal10 := "BK15"."X12-2 SPARE", signal11 := "BK15"."X13-2 SPARE", signal12 := "BK15"."X14-2 SPARE", signal13 := "BK15"."X15-2 SPARE", signal14 := "BK15"."X16-2 SPARE", signal15 := "BK15"."X17-2 SPARE", interfaceSignals := "InstInterfaceSignals".statInterfaceSignalsHmi[17].valueSymbolLeft)
   END_RUNG
   // the same network as SCL:
   #instSignals17Left(signal00 := "BK15"."X10-1 HIPOT&THICKNESS Z-AXIS LIMIT SENSOR(-)",   // "LAF_InterfaceSignalsBool"
                      signal01 := "BK15"."X11-1 HIPOT&THICKNESS Z-AXIS LIMIT SENSOR(+)",
                      signal02 := "BK15"."X12-1 HIPOT&THICKNESS STACK DETECT SENSOR",
                      signal03 := "BK15"."X13-1 HI-POT SAFETY PIN LOADING SENSOR",
                      signal04 := "BK15"."X14-1 SPARE",
                      signal05 := "BK15"."X15-1 SPARE",
                      signal06 := "BK15"."X16-1 SPARE",
                      signal07 := "BK15"."X17-1 SPARE",
                      signal08 := "BK15"."X10-2 HIPOT&THICKNESS Z-AXIS HOME SENSOR",
                      signal09 := "BK15"."X11-2 SPARE",
                      signal10 := "BK15"."X12-2 SPARE",
                      signal11 := "BK15"."X13-2 SPARE",
                      signal12 := "BK15"."X14-2 SPARE",
                      signal13 := "BK15"."X15-2 SPARE",
                      signal14 := "BK15"."X16-2 SPARE",
                      signal15 := "BK15"."X17-2 SPARE",
                      interfaceSignals := "InstInterfaceSignals".statInterfaceSignalsHmi[17].valueSymbolLeft);
END_REGION

REGION Network 23: Interface Signals 18 BK16
   RUNG wire#powerrail
      #instSignals18Left(signal00 := "BK16"."X10-1 FINAL VISION STAGE LIFT UP", signal01 := "BK16"."X10-2 FINAL VISION STAGE LIFT DOWN", signal02 := "BK16"."X12-1 FINAL VISION LIGHT UP", signal03 := "BK16"."X12-2 FINAL VISION LIGHT DOWN", signal04 := "BK16"."X14-1 FINAL VISION STAGE DETECT SENSOR", signal05 := "BK16"."X14-2 SPARE", signal06 := "BK16"."X16-1 SPARE", signal07 := "BK16"."X16-2 SPARE", signal08 :=, signal09 :=, signal10 :=, signal11 :=, signal12 :=, signal13 :=, signal14 :=, signal15 :=, interfaceSignals := "InstInterfaceSignals".statInterfaceSignalsHmi[18].valueSymbolLeft)
   END_RUNG
   // the same network as SCL:
   #instSignals18Left(signal00 := "BK16"."X10-1 FINAL VISION STAGE LIFT UP",   // "LAF_InterfaceSignalsBool"
                      signal01 := "BK16"."X10-2 FINAL VISION STAGE LIFT DOWN",
                      signal02 := "BK16"."X12-1 FINAL VISION LIGHT UP",
                      signal03 := "BK16"."X12-2 FINAL VISION LIGHT DOWN",
                      signal04 := "BK16"."X14-1 FINAL VISION STAGE DETECT SENSOR",
                      signal05 := "BK16"."X14-2 SPARE",
                      signal06 := "BK16"."X16-1 SPARE",
                      signal07 := "BK16"."X16-2 SPARE",
                      interfaceSignals := "InstInterfaceSignals".statInterfaceSignalsHmi[18].valueSymbolLeft);
END_REGION

REGION Network 24: Interface Signals 19 BK17
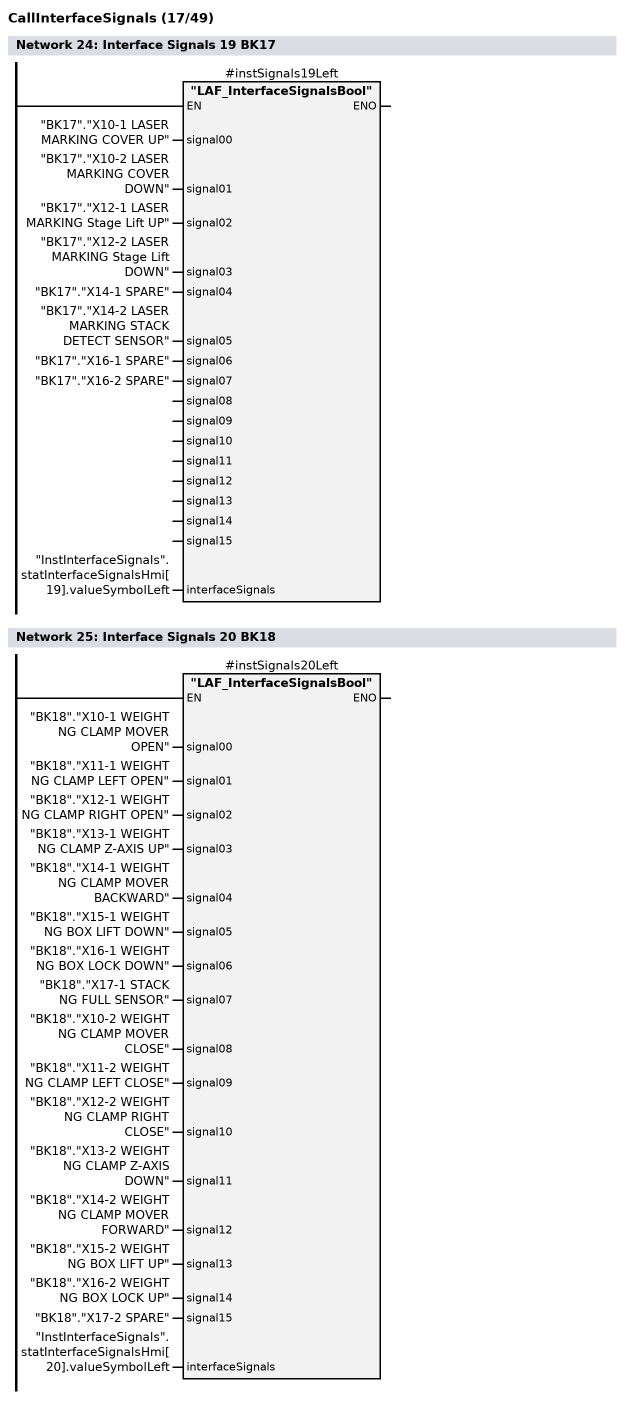
   RUNG wire#powerrail
      #instSignals19Left(signal00 := "BK17"."X10-1 LASER MARKING COVER UP", signal01 := "BK17"."X10-2 LASER MARKING COVER DOWN", signal02 := "BK17"."X12-1 LASER MARKING Stage Lift UP", signal03 := "BK17"."X12-2 LASER MARKING Stage Lift DOWN", signal04 := "BK17"."X14-1 SPARE", signal05 := "BK17"."X14-2 LASER MARKING STACK DETECT SENSOR", signal06 := "BK17"."X16-1 SPARE", signal07 := "BK17"."X16-2 SPARE", signal08 :=, signal09 :=, signal10 :=, signal11 :=, signal12 :=, signal13 :=, signal14 :=, signal15 :=, interfaceSignals := "InstInterfaceSignals".statInterfaceSignalsHmi[19].valueSymbolLeft)
   END_RUNG
   // the same network as SCL:
   #instSignals19Left(signal00 := "BK17"."X10-1 LASER MARKING COVER UP",   // "LAF_InterfaceSignalsBool"
                      signal01 := "BK17"."X10-2 LASER MARKING COVER DOWN",
                      signal02 := "BK17"."X12-1 LASER MARKING Stage Lift UP",
                      signal03 := "BK17"."X12-2 LASER MARKING Stage Lift DOWN",
                      signal04 := "BK17"."X14-1 SPARE",
                      signal05 := "BK17"."X14-2 LASER MARKING STACK DETECT SENSOR",
                      signal06 := "BK17"."X16-1 SPARE",
                      signal07 := "BK17"."X16-2 SPARE",
                      interfaceSignals := "InstInterfaceSignals".statInterfaceSignalsHmi[19].valueSymbolLeft);
END_REGION

REGION Network 25: Interface Signals 20 BK18
   RUNG wire#powerrail
      #instSignals20Left(signal00 := "BK18"."X10-1 WEIGHT NG CLAMP MOVER OPEN", signal01 := "BK18"."X11-1 WEIGHT NG CLAMP LEFT OPEN", signal02 := "BK18"."X12-1 WEIGHT NG CLAMP RIGHT OPEN", signal03 := "BK18"."X13-1 WEIGHT NG CLAMP Z-AXIS UP", signal04 := "BK18"."X14-1 WEIGHT NG CLAMP MOVER BACKWARD", signal05 := "BK18"."X15-1 WEIGHT NG BOX LIFT DOWN", signal06 := "BK18"."X16-1 WEIGHT NG BOX LOCK DOWN", signal07 := "BK18"."X17-1 STACK NG FULL SENSOR", signal08 := "BK18"."X10-2 WEIGHT NG CLAMP MOVER CLOSE", signal09 := "BK18"."X11-2 WEIGHT NG CLAMP LEFT CLOSE", signal10 := "BK18"."X12-2 WEIGHT NG CLAMP RIGHT CLOSE", signal11 := "BK18"."X13-2 WEIGHT NG CLAMP Z-AXIS DOWN", signal12 := "BK18"."X14-2 WEIGHT NG CLAMP MOVER FORWARD", signal13 := "BK18"."X15-2 WEIGHT NG BOX LIFT UP", signal14 := "BK18"."X16-2 WEIGHT NG BOX LOCK UP", signal15 := "BK18"."X17-2 SPARE", interfaceSignals := "InstInterfaceSignals".statInterfaceSignalsHmi[20].valueSymbolLeft)
   END_RUNG
   // the same network as SCL:
   #instSignals20Left(signal00 := "BK18"."X10-1 WEIGHT NG CLAMP MOVER OPEN",   // "LAF_InterfaceSignalsBool"
                      signal01 := "BK18"."X11-1 WEIGHT NG CLAMP LEFT OPEN",
                      signal02 := "BK18"."X12-1 WEIGHT NG CLAMP RIGHT OPEN",
                      signal03 := "BK18"."X13-1 WEIGHT NG CLAMP Z-AXIS UP",
                      signal04 := "BK18"."X14-1 WEIGHT NG CLAMP MOVER BACKWARD",
                      signal05 := "BK18"."X15-1 WEIGHT NG BOX LIFT DOWN",
                      signal06 := "BK18"."X16-1 WEIGHT NG BOX LOCK DOWN",
                      signal07 := "BK18"."X17-1 STACK NG FULL SENSOR",
                      signal08 := "BK18"."X10-2 WEIGHT NG CLAMP MOVER CLOSE",
                      signal09 := "BK18"."X11-2 WEIGHT NG CLAMP LEFT CLOSE",
                      signal10 := "BK18"."X12-2 WEIGHT NG CLAMP RIGHT CLOSE",
                      signal11 := "BK18"."X13-2 WEIGHT NG CLAMP Z-AXIS DOWN",
                      signal12 := "BK18"."X14-2 WEIGHT NG CLAMP MOVER FORWARD",
                      signal13 := "BK18"."X15-2 WEIGHT NG BOX LIFT UP",
                      signal14 := "BK18"."X16-2 WEIGHT NG BOX LOCK UP",
                      signal15 := "BK18"."X17-2 SPARE",
                      interfaceSignals := "InstInterfaceSignals".statInterfaceSignalsHmi[20].valueSymbolLeft);
END_REGION

REGION Network 26: Interface Signals 21 BK19
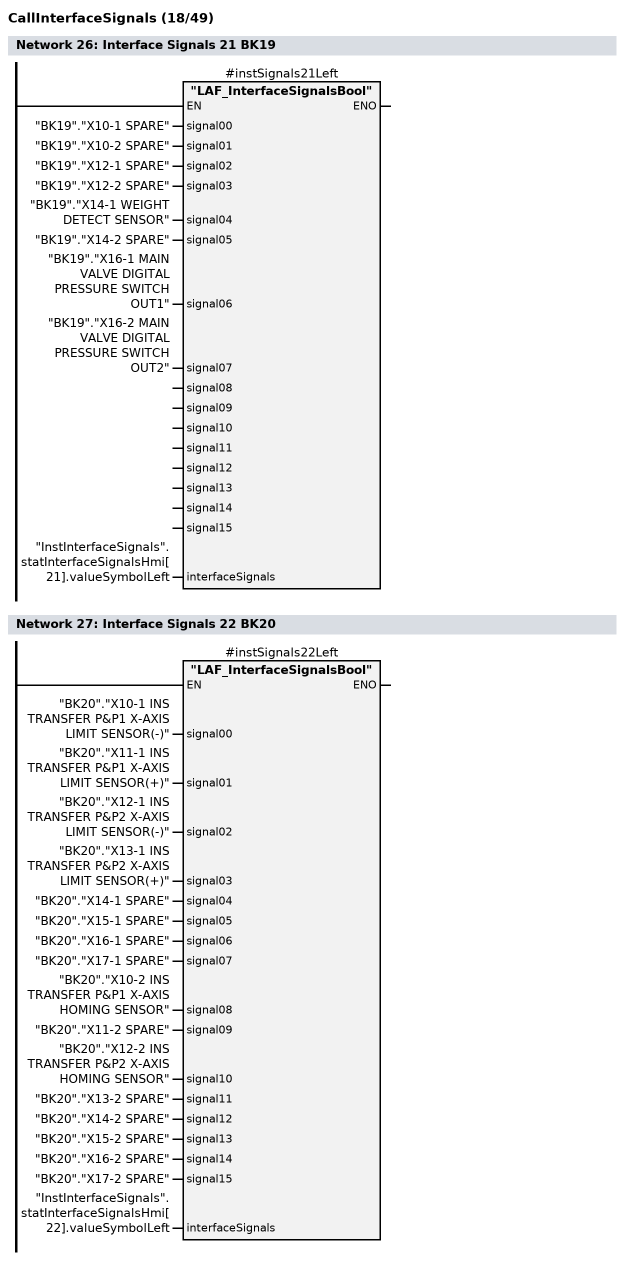
   RUNG wire#powerrail
      #instSignals21Left(signal00 := "BK19"."X10-1 SPARE", signal01 := "BK19"."X10-2 SPARE", signal02 := "BK19"."X12-1 SPARE", signal03 := "BK19"."X12-2 SPARE", signal04 := "BK19"."X14-1 WEIGHT DETECT SENSOR", signal05 := "BK19"."X14-2 SPARE", signal06 := "BK19"."X16-1 MAIN VALVE DIGITAL PRESSURE SWITCH OUT1", signal07 := "BK19"."X16-2 MAIN VALVE DIGITAL PRESSURE SWITCH OUT2", signal08 :=, signal09 :=, signal10 :=, signal11 :=, signal12 :=, signal13 :=, signal14 :=, signal15 :=, interfaceSignals := "InstInterfaceSignals".statInterfaceSignalsHmi[21].valueSymbolLeft)
   END_RUNG
   // the same network as SCL:
   #instSignals21Left(signal00 := "BK19"."X10-1 SPARE",   // "LAF_InterfaceSignalsBool"
                      signal01 := "BK19"."X10-2 SPARE",
                      signal02 := "BK19"."X12-1 SPARE",
                      signal03 := "BK19"."X12-2 SPARE",
                      signal04 := "BK19"."X14-1 WEIGHT DETECT SENSOR",
                      signal05 := "BK19"."X14-2 SPARE",
                      signal06 := "BK19"."X16-1 MAIN VALVE DIGITAL PRESSURE SWITCH OUT1",
                      signal07 := "BK19"."X16-2 MAIN VALVE DIGITAL PRESSURE SWITCH OUT2",
                      interfaceSignals := "InstInterfaceSignals".statInterfaceSignalsHmi[21].valueSymbolLeft);
END_REGION

REGION Network 27: Interface Signals 22 BK20
   RUNG wire#powerrail
      #instSignals22Left(signal00 := "BK20"."X10-1 INS TRANSFER P&P1 X-AXIS LIMIT SENSOR(-)", signal01 := "BK20"."X11-1 INS TRANSFER P&P1 X-AXIS LIMIT SENSOR(+)", signal02 := "BK20"."X12-1 INS TRANSFER P&P2 X-AXIS LIMIT SENSOR(-)", signal03 := "BK20"."X13-1 INS TRANSFER P&P2 X-AXIS LIMIT SENSOR(+)", signal04 := "BK20"."X14-1 SPARE", signal05 := "BK20"."X15-1 SPARE", signal06 := "BK20"."X16-1 SPARE", signal07 := "BK20"."X17-1 SPARE", signal08 := "BK20"."X10-2 INS TRANSFER P&P1 X-AXIS HOMING SENSOR", signal09 := "BK20"."X11-2 SPARE", signal10 := "BK20"."X12-2 INS TRANSFER P&P2 X-AXIS HOMING SENSOR", signal11 := "BK20"."X13-2 SPARE", signal12 := "BK20"."X14-2 SPARE", signal13 := "BK20"."X15-2 SPARE", signal14 := "BK20"."X16-2 SPARE", signal15 := "BK20"."X17-2 SPARE", interfaceSignals := "InstInterfaceSignals".statInterfaceSignalsHmi[22].valueSymbolLeft)
   END_RUNG
   // the same network as SCL:
   #instSignals22Left(signal00 := "BK20"."X10-1 INS TRANSFER P&P1 X-AXIS LIMIT SENSOR(-)",   // "LAF_InterfaceSignalsBool"
                      signal01 := "BK20"."X11-1 INS TRANSFER P&P1 X-AXIS LIMIT SENSOR(+)",
                      signal02 := "BK20"."X12-1 INS TRANSFER P&P2 X-AXIS LIMIT SENSOR(-)",
                      signal03 := "BK20"."X13-1 INS TRANSFER P&P2 X-AXIS LIMIT SENSOR(+)",
                      signal04 := "BK20"."X14-1 SPARE",
                      signal05 := "BK20"."X15-1 SPARE",
                      signal06 := "BK20"."X16-1 SPARE",
                      signal07 := "BK20"."X17-1 SPARE",
                      signal08 := "BK20"."X10-2 INS TRANSFER P&P1 X-AXIS HOMING SENSOR",
                      signal09 := "BK20"."X11-2 SPARE",
                      signal10 := "BK20"."X12-2 INS TRANSFER P&P2 X-AXIS HOMING SENSOR",
                      signal11 := "BK20"."X13-2 SPARE",
                      signal12 := "BK20"."X14-2 SPARE",
                      signal13 := "BK20"."X15-2 SPARE",
                      signal14 := "BK20"."X16-2 SPARE",
                      signal15 := "BK20"."X17-2 SPARE",
                      interfaceSignals := "InstInterfaceSignals".statInterfaceSignalsHmi[22].valueSymbolLeft);
END_REGION

REGION Network 28: Interface Signals 23 BK21
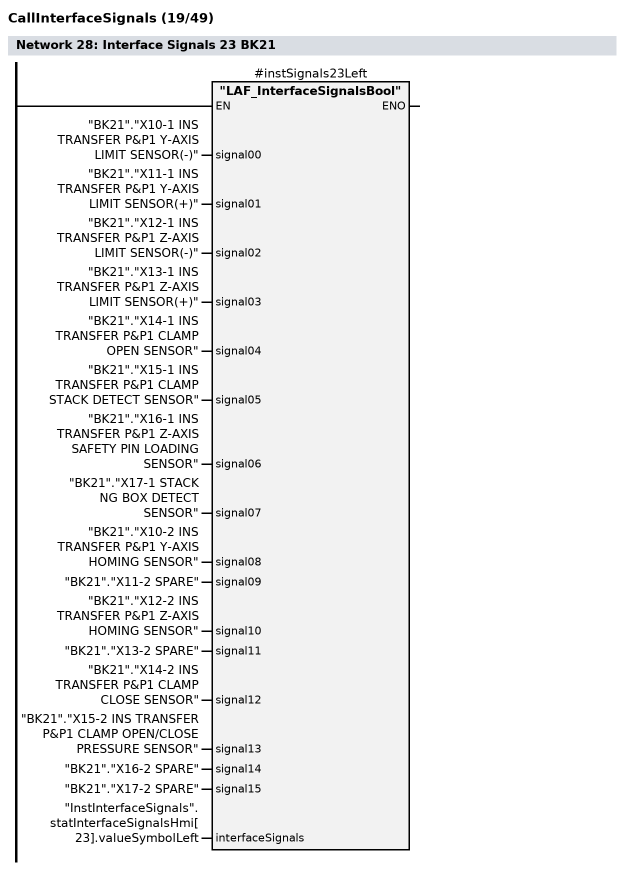
   RUNG wire#powerrail
      #instSignals23Left(signal00 := "BK21"."X10-1 INS TRANSFER P&P1 Y-AXIS LIMIT SENSOR(-)", signal01 := "BK21"."X11-1 INS TRANSFER P&P1 Y-AXIS LIMIT SENSOR(+)", signal02 := "BK21"."X12-1 INS TRANSFER P&P1 Z-AXIS LIMIT SENSOR(-)", signal03 := "BK21"."X13-1 INS TRANSFER P&P1 Z-AXIS LIMIT SENSOR(+)", signal04 := "BK21"."X14-1 INS TRANSFER P&P1 CLAMP OPEN SENSOR", signal05 := "BK21"."X15-1 INS TRANSFER P&P1 CLAMP STACK DETECT SENSOR", signal06 := "BK21"."X16-1 INS TRANSFER P&P1 Z-AXIS SAFETY PIN LOADING SENSOR", signal07 := "BK21"."X17-1 STACK NG BOX DETECT SENSOR", signal08 := "BK21"."X10-2 INS TRANSFER P&P1 Y-AXIS HOMING SENSOR", signal09 := "BK21"."X11-2 SPARE", signal10 := "BK21"."X12-2 INS TRANSFER P&P1 Z-AXIS HOMING SENSOR", signal11 := "BK21"."X13-2 SPARE", signal12 := "BK21"."X14-2 INS TRANSFER P&P1 CLAMP CLOSE SENSOR", signal13 := "BK21"."X15-2 INS TRANSFER P&P1 CLAMP OPEN/CLOSE PRESSURE SENSOR", signal14 := "BK21"."X16-2 SPARE", signal15 := "BK21"."X17-2 SPARE", interfaceSignals := "InstInterfaceSignals".statInterfaceSignalsHmi[23].valueSymbolLeft)
   END_RUNG
   // the same network as SCL:
   #instSignals23Left(signal00 := "BK21"."X10-1 INS TRANSFER P&P1 Y-AXIS LIMIT SENSOR(-)",   // "LAF_InterfaceSignalsBool"
                      signal01 := "BK21"."X11-1 INS TRANSFER P&P1 Y-AXIS LIMIT SENSOR(+)",
                      signal02 := "BK21"."X12-1 INS TRANSFER P&P1 Z-AXIS LIMIT SENSOR(-)",
                      signal03 := "BK21"."X13-1 INS TRANSFER P&P1 Z-AXIS LIMIT SENSOR(+)",
                      signal04 := "BK21"."X14-1 INS TRANSFER P&P1 CLAMP OPEN SENSOR",
                      signal05 := "BK21"."X15-1 INS TRANSFER P&P1 CLAMP STACK DETECT SENSOR",
                      signal06 := "BK21"."X16-1 INS TRANSFER P&P1 Z-AXIS SAFETY PIN LOADING SENSOR",
                      signal07 := "BK21"."X17-1 STACK NG BOX DETECT SENSOR",
                      signal08 := "BK21"."X10-2 INS TRANSFER P&P1 Y-AXIS HOMING SENSOR",
                      signal09 := "BK21"."X11-2 SPARE",
                      signal10 := "BK21"."X12-2 INS TRANSFER P&P1 Z-AXIS HOMING SENSOR",
                      signal11 := "BK21"."X13-2 SPARE",
                      signal12 := "BK21"."X14-2 INS TRANSFER P&P1 CLAMP CLOSE SENSOR",
                      signal13 := "BK21"."X15-2 INS TRANSFER P&P1 CLAMP OPEN/CLOSE PRESSURE SENSOR",
                      signal14 := "BK21"."X16-2 SPARE",
                      signal15 := "BK21"."X17-2 SPARE",
                      interfaceSignals := "InstInterfaceSignals".statInterfaceSignalsHmi[23].valueSymbolLeft);
END_REGION

REGION Network 29: Interface Signals 24 BK22
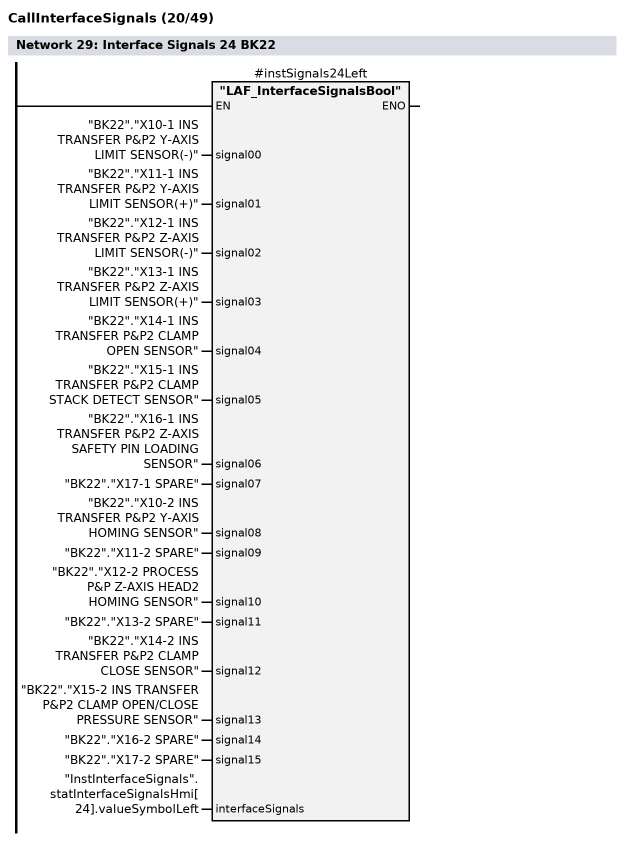
   RUNG wire#powerrail
      #instSignals24Left(signal00 := "BK22"."X10-1 INS TRANSFER P&P2 Y-AXIS LIMIT SENSOR(-)", signal01 := "BK22"."X11-1 INS TRANSFER P&P2 Y-AXIS LIMIT SENSOR(+)", signal02 := "BK22"."X12-1 INS TRANSFER P&P2 Z-AXIS LIMIT SENSOR(-)", signal03 := "BK22"."X13-1 INS TRANSFER P&P2 Z-AXIS LIMIT SENSOR(+)", signal04 := "BK22"."X14-1 INS TRANSFER P&P2 CLAMP OPEN SENSOR", signal05 := "BK22"."X15-1 INS TRANSFER P&P2 CLAMP STACK DETECT SENSOR", signal06 := "BK22"."X16-1 INS TRANSFER P&P2 Z-AXIS SAFETY PIN LOADING SENSOR", signal07 := "BK22"."X17-1 SPARE", signal08 := "BK22"."X10-2 INS TRANSFER P&P2 Y-AXIS HOMING SENSOR", signal09 := "BK22"."X11-2 SPARE", signal10 := "BK22"."X12-2 PROCESS P&P Z-AXIS HEAD2 HOMING SENSOR", signal11 := "BK22"."X13-2 SPARE", signal12 := "BK22"."X14-2 INS TRANSFER P&P2 CLAMP CLOSE SENSOR", signal13 := "BK22"."X15-2 INS TRANSFER P&P2 CLAMP OPEN/CLOSE PRESSURE SENSOR", signal14 := "BK22"."X16-2 SPARE", signal15 := "BK22"."X17-2 SPARE", interfaceSignals := "InstInterfaceSignals".statInterfaceSignalsHmi[24].valueSymbolLeft)
   END_RUNG
   // the same network as SCL:
   #instSignals24Left(signal00 := "BK22"."X10-1 INS TRANSFER P&P2 Y-AXIS LIMIT SENSOR(-)",   // "LAF_InterfaceSignalsBool"
                      signal01 := "BK22"."X11-1 INS TRANSFER P&P2 Y-AXIS LIMIT SENSOR(+)",
                      signal02 := "BK22"."X12-1 INS TRANSFER P&P2 Z-AXIS LIMIT SENSOR(-)",
                      signal03 := "BK22"."X13-1 INS TRANSFER P&P2 Z-AXIS LIMIT SENSOR(+)",
                      signal04 := "BK22"."X14-1 INS TRANSFER P&P2 CLAMP OPEN SENSOR",
                      signal05 := "BK22"."X15-1 INS TRANSFER P&P2 CLAMP STACK DETECT SENSOR",
                      signal06 := "BK22"."X16-1 INS TRANSFER P&P2 Z-AXIS SAFETY PIN LOADING SENSOR",
                      signal07 := "BK22"."X17-1 SPARE",
                      signal08 := "BK22"."X10-2 INS TRANSFER P&P2 Y-AXIS HOMING SENSOR",
                      signal09 := "BK22"."X11-2 SPARE",
                      signal10 := "BK22"."X12-2 PROCESS P&P Z-AXIS HEAD2 HOMING SENSOR",
                      signal11 := "BK22"."X13-2 SPARE",
                      signal12 := "BK22"."X14-2 INS TRANSFER P&P2 CLAMP CLOSE SENSOR",
                      signal13 := "BK22"."X15-2 INS TRANSFER P&P2 CLAMP OPEN/CLOSE PRESSURE SENSOR",
                      signal14 := "BK22"."X16-2 SPARE",
                      signal15 := "BK22"."X17-2 SPARE",
                      interfaceSignals := "InstInterfaceSignals".statInterfaceSignalsHmi[24].valueSymbolLeft);
END_REGION

REGION Network 30: Interface Signals 25 BK23
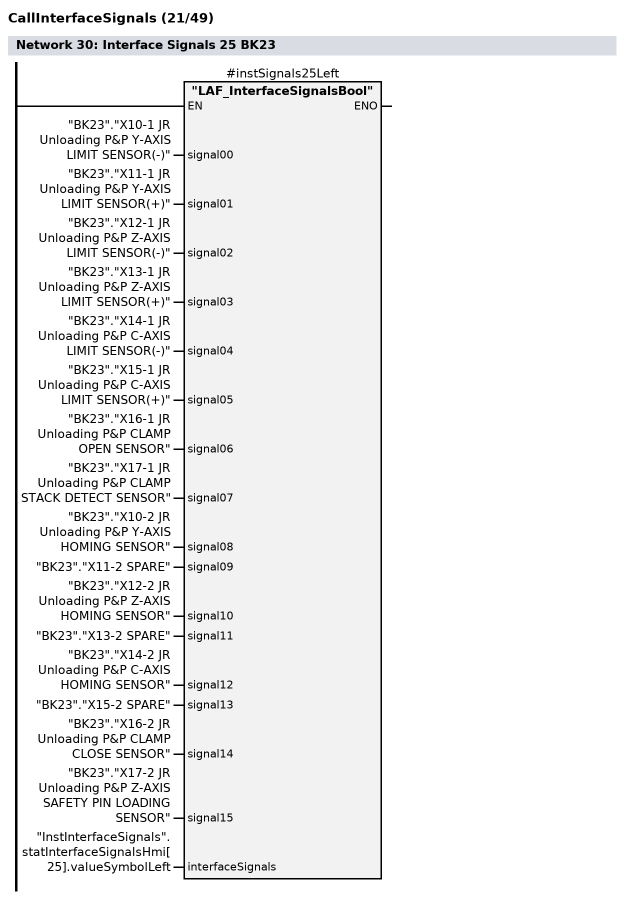
   RUNG wire#powerrail
      #instSignals25Left(signal00 := "BK23"."X10-1 JR Unloading P&P Y-AXIS LIMIT SENSOR(-)", signal01 := "BK23"."X11-1 JR Unloading P&P Y-AXIS LIMIT SENSOR(+)", signal02 := "BK23"."X12-1 JR Unloading P&P Z-AXIS LIMIT SENSOR(-)", signal03 := "BK23"."X13-1 JR Unloading P&P Z-AXIS LIMIT SENSOR(+)", signal04 := "BK23"."X14-1 JR Unloading P&P C-AXIS LIMIT SENSOR(-)", signal05 := "BK23"."X15-1 JR Unloading P&P C-AXIS LIMIT SENSOR(+)", signal06 := "BK23"."X16-1 JR Unloading P&P CLAMP OPEN SENSOR", signal07 := "BK23"."X17-1 JR Unloading P&P CLAMP STACK DETECT SENSOR", signal08 := "BK23"."X10-2 JR Unloading P&P Y-AXIS HOMING SENSOR", signal09 := "BK23"."X11-2 SPARE", signal10 := "BK23"."X12-2 JR Unloading P&P Z-AXIS HOMING SENSOR", signal11 := "BK23"."X13-2 SPARE", signal12 := "BK23"."X14-2 JR Unloading P&P C-AXIS HOMING SENSOR", signal13 := "BK23"."X15-2 SPARE", signal14 := "BK23"."X16-2 JR Unloading P&P CLAMP CLOSE SENSOR", signal15 := "BK23"."X17-2 JR Unloading P&P Z-AXIS SAFETY PIN LOADING SENSOR", interfaceSignals := "InstInterfaceSignals".statInterfaceSignalsHmi[25].valueSymbolLeft)
   END_RUNG
   // the same network as SCL:
   #instSignals25Left(signal00 := "BK23"."X10-1 JR Unloading P&P Y-AXIS LIMIT SENSOR(-)",   // "LAF_InterfaceSignalsBool"
                      signal01 := "BK23"."X11-1 JR Unloading P&P Y-AXIS LIMIT SENSOR(+)",
                      signal02 := "BK23"."X12-1 JR Unloading P&P Z-AXIS LIMIT SENSOR(-)",
                      signal03 := "BK23"."X13-1 JR Unloading P&P Z-AXIS LIMIT SENSOR(+)",
                      signal04 := "BK23"."X14-1 JR Unloading P&P C-AXIS LIMIT SENSOR(-)",
                      signal05 := "BK23"."X15-1 JR Unloading P&P C-AXIS LIMIT SENSOR(+)",
                      signal06 := "BK23"."X16-1 JR Unloading P&P CLAMP OPEN SENSOR",
                      signal07 := "BK23"."X17-1 JR Unloading P&P CLAMP STACK DETECT SENSOR",
                      signal08 := "BK23"."X10-2 JR Unloading P&P Y-AXIS HOMING SENSOR",
                      signal09 := "BK23"."X11-2 SPARE",
                      signal10 := "BK23"."X12-2 JR Unloading P&P Z-AXIS HOMING SENSOR",
                      signal11 := "BK23"."X13-2 SPARE",
                      signal12 := "BK23"."X14-2 JR Unloading P&P C-AXIS HOMING SENSOR",
                      signal13 := "BK23"."X15-2 SPARE",
                      signal14 := "BK23"."X16-2 JR Unloading P&P CLAMP CLOSE SENSOR",
                      signal15 := "BK23"."X17-2 JR Unloading P&P Z-AXIS SAFETY PIN LOADING SENSOR",
                      interfaceSignals := "InstInterfaceSignals".statInterfaceSignalsHmi[25].valueSymbolLeft);
END_REGION

REGION Network 31: Interface Signals 26 BK24
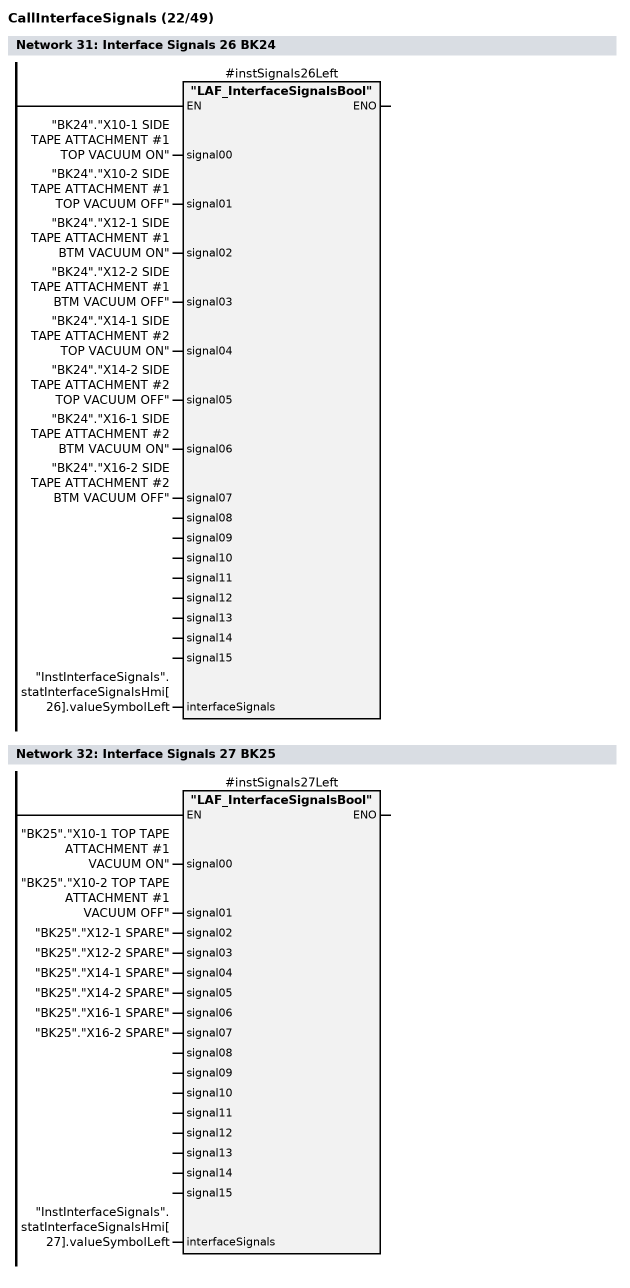
   RUNG wire#powerrail
      #instSignals26Left(signal00 := "BK24"."X10-1 SIDE TAPE ATTACHMENT #1 TOP VACUUM ON", signal01 := "BK24"."X10-2 SIDE TAPE ATTACHMENT #1 TOP VACUUM OFF", signal02 := "BK24"."X12-1 SIDE TAPE ATTACHMENT #1 BTM VACUUM ON", signal03 := "BK24"."X12-2 SIDE TAPE ATTACHMENT #1 BTM VACUUM OFF", signal04 := "BK24"."X14-1 SIDE TAPE ATTACHMENT #2 TOP VACUUM ON", signal05 := "BK24"."X14-2 SIDE TAPE ATTACHMENT #2 TOP VACUUM OFF", signal06 := "BK24"."X16-1 SIDE TAPE ATTACHMENT #2 BTM VACUUM ON", signal07 := "BK24"."X16-2 SIDE TAPE ATTACHMENT #2 BTM VACUUM OFF", signal08 :=, signal09 :=, signal10 :=, signal11 :=, signal12 :=, signal13 :=, signal14 :=, signal15 :=, interfaceSignals := "InstInterfaceSignals".statInterfaceSignalsHmi[26].valueSymbolLeft)
   END_RUNG
   // the same network as SCL:
   #instSignals26Left(signal00 := "BK24"."X10-1 SIDE TAPE ATTACHMENT #1 TOP VACUUM ON",   // "LAF_InterfaceSignalsBool"
                      signal01 := "BK24"."X10-2 SIDE TAPE ATTACHMENT #1 TOP VACUUM OFF",
                      signal02 := "BK24"."X12-1 SIDE TAPE ATTACHMENT #1 BTM VACUUM ON",
                      signal03 := "BK24"."X12-2 SIDE TAPE ATTACHMENT #1 BTM VACUUM OFF",
                      signal04 := "BK24"."X14-1 SIDE TAPE ATTACHMENT #2 TOP VACUUM ON",
                      signal05 := "BK24"."X14-2 SIDE TAPE ATTACHMENT #2 TOP VACUUM OFF",
                      signal06 := "BK24"."X16-1 SIDE TAPE ATTACHMENT #2 BTM VACUUM ON",
                      signal07 := "BK24"."X16-2 SIDE TAPE ATTACHMENT #2 BTM VACUUM OFF",
                      interfaceSignals := "InstInterfaceSignals".statInterfaceSignalsHmi[26].valueSymbolLeft);
END_REGION

REGION Network 32: Interface Signals 27 BK25
   RUNG wire#powerrail
      #instSignals27Left(signal00 := "BK25"."X10-1 TOP TAPE ATTACHMENT #1 VACUUM ON", signal01 := "BK25"."X10-2 TOP TAPE ATTACHMENT #1 VACUUM OFF", signal02 := "BK25"."X12-1 SPARE", signal03 := "BK25"."X12-2 SPARE", signal04 := "BK25"."X14-1 SPARE", signal05 := "BK25"."X14-2 SPARE", signal06 := "BK25"."X16-1 SPARE", signal07 := "BK25"."X16-2 SPARE", signal08 :=, signal09 :=, signal10 :=, signal11 :=, signal12 :=, signal13 :=, signal14 :=, signal15 :=, interfaceSignals := "InstInterfaceSignals".statInterfaceSignalsHmi[27].valueSymbolLeft)
   END_RUNG
   // the same network as SCL:
   #instSignals27Left(signal00 := "BK25"."X10-1 TOP TAPE ATTACHMENT #1 VACUUM ON",   // "LAF_InterfaceSignalsBool"
                      signal01 := "BK25"."X10-2 TOP TAPE ATTACHMENT #1 VACUUM OFF",
                      signal02 := "BK25"."X12-1 SPARE",
                      signal03 := "BK25"."X12-2 SPARE",
                      signal04 := "BK25"."X14-1 SPARE",
                      signal05 := "BK25"."X14-2 SPARE",
                      signal06 := "BK25"."X16-1 SPARE",
                      signal07 := "BK25"."X16-2 SPARE",
                      interfaceSignals := "InstInterfaceSignals".statInterfaceSignalsHmi[27].valueSymbolLeft);
END_REGION

REGION Network 33: Interface Signals 28 PM01
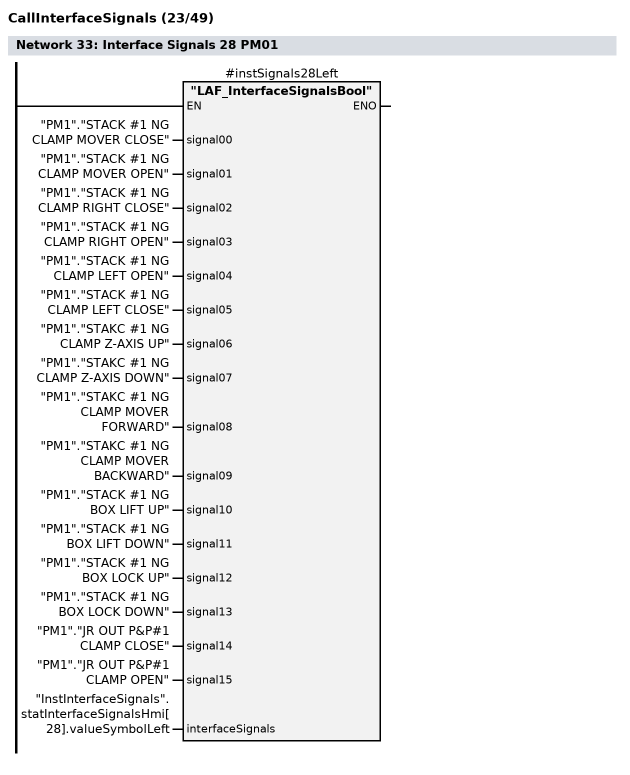
   RUNG wire#powerrail
      #instSignals28Left(signal00 := "PM1"."STACK #1 NG CLAMP MOVER CLOSE", signal01 := "PM1"."STACK #1 NG CLAMP MOVER OPEN", signal02 := "PM1"."STACK #1 NG CLAMP RIGHT CLOSE", signal03 := "PM1"."STACK #1 NG CLAMP RIGHT OPEN", signal04 := "PM1"."STACK #1 NG CLAMP LEFT OPEN", signal05 := "PM1"."STACK #1 NG CLAMP LEFT CLOSE", signal06 := "PM1"."STAKC #1 NG CLAMP Z-AXIS UP", signal07 := "PM1"."STAKC #1 NG CLAMP Z-AXIS DOWN", signal08 := "PM1"."STAKC #1 NG CLAMP MOVER FORWARD", signal09 := "PM1"."STAKC #1 NG CLAMP MOVER BACKWARD", signal10 := "PM1"."STACK #1 NG BOX LIFT UP", signal11 := "PM1"."STACK #1 NG BOX LIFT DOWN", signal12 := "PM1"."STACK #1 NG BOX LOCK UP", signal13 := "PM1"."STACK #1 NG BOX LOCK DOWN", signal14 := "PM1"."JR OUT P&P#1 CLAMP CLOSE", signal15 := "PM1"."JR OUT P&P#1 CLAMP OPEN", interfaceSignals := "InstInterfaceSignals".statInterfaceSignalsHmi[28].valueSymbolLeft)
   END_RUNG
   // the same network as SCL:
   #instSignals28Left(signal00 := "PM1"."STACK #1 NG CLAMP MOVER CLOSE",   // "LAF_InterfaceSignalsBool"
                      signal01 := "PM1"."STACK #1 NG CLAMP MOVER OPEN",
                      signal02 := "PM1"."STACK #1 NG CLAMP RIGHT CLOSE",
                      signal03 := "PM1"."STACK #1 NG CLAMP RIGHT OPEN",
                      signal04 := "PM1"."STACK #1 NG CLAMP LEFT OPEN",
                      signal05 := "PM1"."STACK #1 NG CLAMP LEFT CLOSE",
                      signal06 := "PM1"."STAKC #1 NG CLAMP Z-AXIS UP",
                      signal07 := "PM1"."STAKC #1 NG CLAMP Z-AXIS DOWN",
                      signal08 := "PM1"."STAKC #1 NG CLAMP MOVER FORWARD",
                      signal09 := "PM1"."STAKC #1 NG CLAMP MOVER BACKWARD",
                      signal10 := "PM1"."STACK #1 NG BOX LIFT UP",
                      signal11 := "PM1"."STACK #1 NG BOX LIFT DOWN",
                      signal12 := "PM1"."STACK #1 NG BOX LOCK UP",
                      signal13 := "PM1"."STACK #1 NG BOX LOCK DOWN",
                      signal14 := "PM1"."JR OUT P&P#1 CLAMP CLOSE",
                      signal15 := "PM1"."JR OUT P&P#1 CLAMP OPEN",
                      interfaceSignals := "InstInterfaceSignals".statInterfaceSignalsHmi[28].valueSymbolLeft);
END_REGION

REGION Network 34: Interface Signals 29 PM02
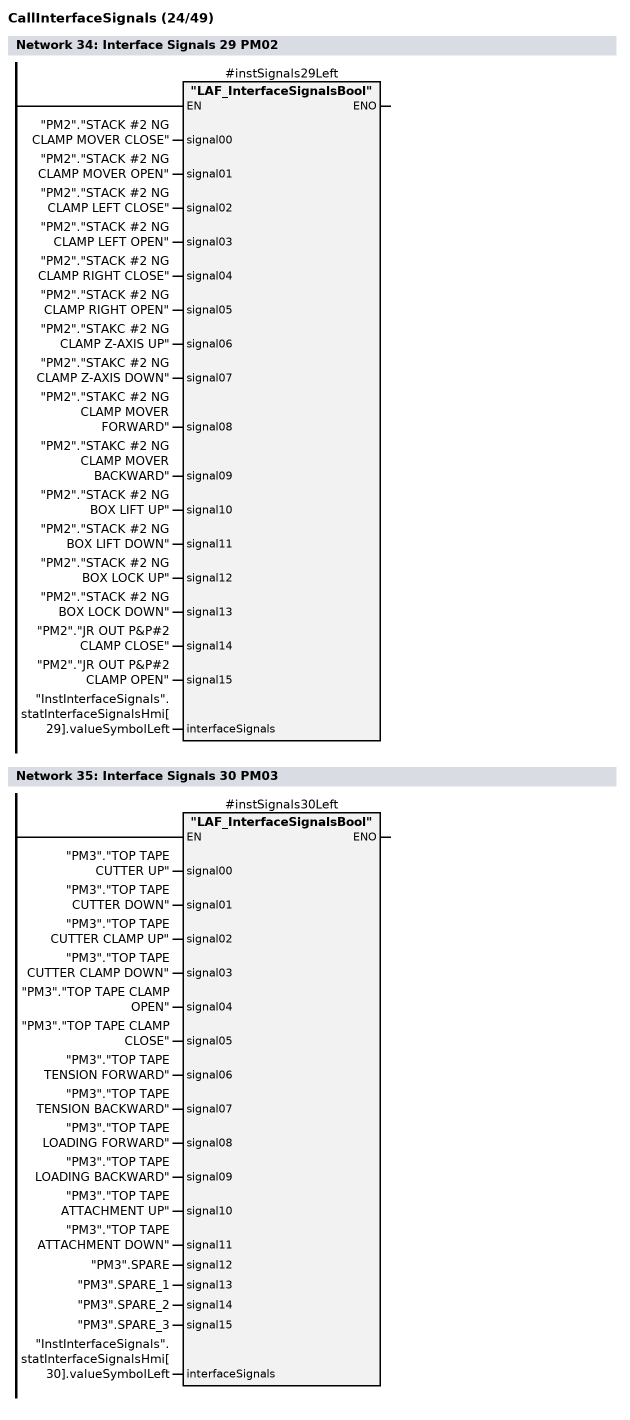
   RUNG wire#powerrail
      #instSignals29Left(signal00 := "PM2"."STACK #2 NG CLAMP MOVER CLOSE", signal01 := "PM2"."STACK #2 NG CLAMP MOVER OPEN", signal02 := "PM2"."STACK #2 NG CLAMP LEFT CLOSE", signal03 := "PM2"."STACK #2 NG CLAMP LEFT OPEN", signal04 := "PM2"."STACK #2 NG CLAMP RIGHT CLOSE", signal05 := "PM2"."STACK #2 NG CLAMP RIGHT OPEN", signal06 := "PM2"."STAKC #2 NG CLAMP Z-AXIS UP", signal07 := "PM2"."STAKC #2 NG CLAMP Z-AXIS DOWN", signal08 := "PM2"."STAKC #2 NG CLAMP MOVER FORWARD", signal09 := "PM2"."STAKC #2 NG CLAMP MOVER BACKWARD", signal10 := "PM2"."STACK #2 NG BOX LIFT UP", signal11 := "PM2"."STACK #2 NG BOX LIFT DOWN", signal12 := "PM2"."STACK #2 NG BOX LOCK UP", signal13 := "PM2"."STACK #2 NG BOX LOCK DOWN", signal14 := "PM2"."JR OUT P&P#2 CLAMP CLOSE", signal15 := "PM2"."JR OUT P&P#2 CLAMP OPEN", interfaceSignals := "InstInterfaceSignals".statInterfaceSignalsHmi[29].valueSymbolLeft)
   END_RUNG
   // the same network as SCL:
   #instSignals29Left(signal00 := "PM2"."STACK #2 NG CLAMP MOVER CLOSE",   // "LAF_InterfaceSignalsBool"
                      signal01 := "PM2"."STACK #2 NG CLAMP MOVER OPEN",
                      signal02 := "PM2"."STACK #2 NG CLAMP LEFT CLOSE",
                      signal03 := "PM2"."STACK #2 NG CLAMP LEFT OPEN",
                      signal04 := "PM2"."STACK #2 NG CLAMP RIGHT CLOSE",
                      signal05 := "PM2"."STACK #2 NG CLAMP RIGHT OPEN",
                      signal06 := "PM2"."STAKC #2 NG CLAMP Z-AXIS UP",
                      signal07 := "PM2"."STAKC #2 NG CLAMP Z-AXIS DOWN",
                      signal08 := "PM2"."STAKC #2 NG CLAMP MOVER FORWARD",
                      signal09 := "PM2"."STAKC #2 NG CLAMP MOVER BACKWARD",
                      signal10 := "PM2"."STACK #2 NG BOX LIFT UP",
                      signal11 := "PM2"."STACK #2 NG BOX LIFT DOWN",
                      signal12 := "PM2"."STACK #2 NG BOX LOCK UP",
                      signal13 := "PM2"."STACK #2 NG BOX LOCK DOWN",
                      signal14 := "PM2"."JR OUT P&P#2 CLAMP CLOSE",
                      signal15 := "PM2"."JR OUT P&P#2 CLAMP OPEN",
                      interfaceSignals := "InstInterfaceSignals".statInterfaceSignalsHmi[29].valueSymbolLeft);
END_REGION

REGION Network 35: Interface Signals 30 PM03
   RUNG wire#powerrail
      #instSignals30Left(signal00 := "PM3"."TOP TAPE CUTTER UP", signal01 := "PM3"."TOP TAPE CUTTER DOWN", signal02 := "PM3"."TOP TAPE CUTTER CLAMP UP", signal03 := "PM3"."TOP TAPE CUTTER CLAMP DOWN", signal04 := "PM3"."TOP TAPE CLAMP OPEN", signal05 := "PM3"."TOP TAPE CLAMP CLOSE", signal06 := "PM3"."TOP TAPE TENSION FORWARD", signal07 := "PM3"."TOP TAPE TENSION BACKWARD", signal08 := "PM3"."TOP TAPE LOADING FORWARD", signal09 := "PM3"."TOP TAPE LOADING BACKWARD", signal10 := "PM3"."TOP TAPE ATTACHMENT UP", signal11 := "PM3"."TOP TAPE ATTACHMENT DOWN", signal12 := "PM3".SPARE, signal13 := "PM3".SPARE_1, signal14 := "PM3".SPARE_2, signal15 := "PM3".SPARE_3, interfaceSignals := "InstInterfaceSignals".statInterfaceSignalsHmi[30].valueSymbolLeft)
   END_RUNG
   // the same network as SCL:
   #instSignals30Left(signal00 := "PM3"."TOP TAPE CUTTER UP",   // "LAF_InterfaceSignalsBool"
                      signal01 := "PM3"."TOP TAPE CUTTER DOWN",
                      signal02 := "PM3"."TOP TAPE CUTTER CLAMP UP",
                      signal03 := "PM3"."TOP TAPE CUTTER CLAMP DOWN",
                      signal04 := "PM3"."TOP TAPE CLAMP OPEN",
                      signal05 := "PM3"."TOP TAPE CLAMP CLOSE",
                      signal06 := "PM3"."TOP TAPE TENSION FORWARD",
                      signal07 := "PM3"."TOP TAPE TENSION BACKWARD",
                      signal08 := "PM3"."TOP TAPE LOADING FORWARD",
                      signal09 := "PM3"."TOP TAPE LOADING BACKWARD",
                      signal10 := "PM3"."TOP TAPE ATTACHMENT UP",
                      signal11 := "PM3"."TOP TAPE ATTACHMENT DOWN",
                      signal12 := "PM3".SPARE,
                      signal13 := "PM3".SPARE_1,
                      signal14 := "PM3".SPARE_2,
                      signal15 := "PM3".SPARE_3,
                      interfaceSignals := "InstInterfaceSignals".statInterfaceSignalsHmi[30].valueSymbolLeft);
END_REGION

REGION Network 36: Interface Signals 31 PM04
